# B&R Automation Studio project 8238 (part 17)

#### _GetRights.st - Ermittelt Lese- und Schreibrecht
```iecst
(********************************************************************
 * COPYRIGHT -- Herbert Kannegiesser GmbH
 ********************************************************************
 * Program: mnParam
 * File: _GetRights.st
 * Author: hunholz
 * Created: February 20, 2012
 ********************************************************************
 * Implementation of program mnParam
 ********************************************************************)

(* Ermittelt Lese- und Schreibrecht *)
FUNCTION_BLOCK _GetRights

	IF Enable THEN

		Status := ERR_OK;

		bWriteAccess := 0;
		bReadAccess := 0;

		IF lPtrLogicStruct = 0 THEN

			Status := MNPARAM_STAT_NULLPOINTER;
			RETURN;

		END_IF

		_DoLogStruc ACCESS lPtrLogicStruct;

		IF siWriteAccess >= 0 THEN

			bWriteAccess := SINT_TO_USINT(siWriteAccess);

		ELSE

			_wLogIdx := wReference;
			_xReady := FALSE;
			_bSearchIt := 0;

			REPEAT

				IF _wLogIdx <= wMaxIdxLogicStruct  AND _wLogIdx > 0 THEN

					IF _DoLogStruc.LogicalStruct[_wLogIdx].siWriteAccess >= 0 THEN

						// Gültiges Recht gefunden
						bWriteAccess := SINT_TO_USINT(_DoLogStruc.LogicalStruct[_wLogIdx].siWriteAccess);
						_xReady := TRUE;

					ELSE

						IF _DoLogStruc.LogicalStruct[_wLogIdx].iReferenz > 0 THEN

							_wLogIdx := INT_TO_UINT(_DoLogStruc.LogicalStruct[_wLogIdx].iReferenz);
							_bSearchIt := _bSearchIt + 1;

							// Wenn maximale Suchtiefe erreicht, dann abbrechen
							_xReady := _bSearchIt > 6;

						ELSE

							// Kein Recht definiert und Referenz verweist auf Container, abbrechen
							_xReady := TRUE;

						END_IF

					END_IF

				ELSE

					// Referenz ist ungültig, abbrechen
					_xReady := TRUE;

				END_IF

				UNTIL
					_xReady
			END_REPEAT

		END_IF

		IF siReadAccess >= 0 THEN

			bReadAccess := SINT_TO_USINT(siReadAccess);

		ELSE

			_wLogIdx := wReference;
			_xReady := FALSE;
			_bSearchIt := 0;

			REPEAT

				IF _wLogIdx <= wMaxIdxLogicStruct  AND _wLogIdx > 0 THEN

					IF _DoLogStruc.LogicalStruct[_wLogIdx].siVisibleAccess >= 0 THEN

						// Gültiges Recht gefunden
						bReadAccess := SINT_TO_USINT(_DoLogStruc.LogicalStruct[_wLogIdx].siVisibleAccess);
						_xReady := TRUE;

					ELSE

						IF _DoLogStruc.LogicalStruct[_wLogIdx].iReferenz > 0 THEN

							_wLogIdx := INT_TO_UINT(_DoLogStruc.LogicalStruct[_wLogIdx].iReferenz);
							_bSearchIt := _bSearchIt + 1;

							// Wenn maximale Suchtiefe erreicht, dann abbrechen
							_xReady := _bSearchIt > 6;

						ELSE

							// Kein Recht definiert und Referenz verweist auf Container, abbrechen
							_xReady := TRUE;

						END_IF

					END_IF

				ELSE

					// Referenz ist ungültig, abbrechen
					_xReady := TRUE;

				END_IF

				UNTIL
				_xReady
			END_REPEAT

		END_IF

	ELSE

		Status := ERR_FUB_ENABLE_FALSE;

	END_IF

END_FUNCTION_BLOCK
```

#### _BinSearchTxtLine.st - Finde Textzeile nach Function-ID und Nummer
```iecst
(********************************************************************
 * COPYRIGHT -- Herbert Kannegiesser GmbH
 ********************************************************************
 * Program: mnParam
 * File: _BinSearchTxtLine.st
 * Author: hunholz
 * Created: February 21, 2012
 ********************************************************************
 * Implementation of program mnParam
 ********************************************************************)

(* Finde Textzeile nach Function-ID und Nummer *)
FUNCTION _BinSearchTxtLine

	_BinSearchTxtLine := 65535;

	IF lPtrTxtLines = 0 OR wCntRows < 1 THEN
		// Null-Pointer oder leere Liste
		RETURN;
	END_IF

	// Access auf dynamische Struktur
	_pTextLines ACCESS lPtrTxtLines;

	_wMin := 0;
	_wMax := wCntRows-1;

	WHILE TRUE DO

		IF (_wMin <= _wMax) THEN

			// Suche nach korrektem IdxPar
			// Middle Index berechnen
			_wMid := (_wMin + _wMax) / 2;

			// Suche erfolgreich?
			IF _pTextLines[_wMid].wFunctionID = wFunctionID THEN

				IF _pTextLines[_wMid].wNumber = wNo THEN

					_BinSearchTxtLine := _wMid;

					EXIT;

				ELSIF wNo < _pTextLines[_wMid].wNumber THEN

					_wMax := _wMid - 1;

				ELSE

					_wMin := _wMid + 1;

				END_IF

			ELSIF wFunctionID < _pTextLines[_wMid].wFunctionID THEN

				_wMax := _wMid - 1;

			ELSE

				_wMin := _wMid + 1;

			END_IF

		ELSE
			// Fehler in der Binären-Suche
			// zB entsprechende Zeile konnte nicht gefunden werden
			EXIT;
		END_IF;

	END_WHILE;

END_FUNCTION
```

#### _BinSearchHlpTxtLine.st - Finde Hilfstextzeile nach Funktion-ID und Nummer
```iecst
(********************************************************************
 * COPYRIGHT -- Herbert Kannegiesser GmbH
 ********************************************************************
 * Program: mnParam
 * File: _BinSearchHlpTxtLine.st
 * Author: hunholz
 * Created: February 21, 2012
 ********************************************************************
 * Implementation of program mnParam
 ********************************************************************)

(* Finde Hilfstextzeile nach Funktion-ID und Nummer *)
FUNCTION _BinSearchHlpTxtLine

	_BinSearchHlpTxtLine := 65535;

	IF lPtrHlpTxtLines = 0 OR wCntRows < 1 THEN
		// Null-Pointer oder leere Liste
		RETURN;
	END_IF

	// Access auf dynamische Struktur
	_pHlpTextLines ACCESS lPtrHlpTxtLines;

	_wMin := 0;
	_wMax := wCntRows-1;

	WHILE TRUE DO

		IF (_wMin <= _wMax) THEN

			// Suche nach korrektem IdxPar
			// Middle Index berechnen
			_wMid := (_wMin + _wMax) / 2;

			// Suche erfolgreich?
			IF _pHlpTextLines[_wMid].wFunctionID = wFunctionID THEN

				IF _pHlpTextLines[_wMid].wNumber = wNo THEN

					_BinSearchHlpTxtLine := _wMid;

					EXIT;

				ELSIF wNo < _pHlpTextLines[_wMid].wNumber THEN

					_wMax := _wMid - 1;

				ELSE

					_wMin := _wMid + 1;

				END_IF

			ELSIF wFunctionID < _pHlpTextLines[_wMid].wFunctionID THEN

				_wMax := _wMid - 1;

			ELSE

				_wMin := _wMid + 1;

			END_IF

		ELSE
			// Fehler in der Binären-Suche
			// zB entsprechende Zeile konnte nicht gefunden werden
			EXIT;
		END_IF;

	END_WHILE;

END_FUNCTION
```

#### _LimParam.st - Parameter begrenzen
```iecst
(********************************************************************
 * COPYRIGHT -- Herbert Kannegiesser GmbH
 ********************************************************************
 * Program: mnParam
 * File: _LimParam.st
 * Author: hunholz
 * Created: June 12, 2012
 ********************************************************************
 * Implementation of program mnParam
 ********************************************************************)

(* Parameter begrenzen *)
FUNCTION_BLOCK _LimParam

	IF pParamNum = 0 OR pCsvNumRow = 0 THEN

		RETURN;

	END_IF

	_ParamNum ACCESS pParamNum;
	_CsvNumRow ACCESS pCsvNumRow;

	IF _CsvNumRow.bRowType = 10 THEN

		_CsvNumRow.diValue := LIMIT(_ParamNum.diMinValue, _CsvNumRow.diValue, _ParamNum.diMaxValue);

	ELSE

		_rValue ACCESS ADR(_CsvNumRow.diValue);
		_rMinValue ACCESS ADR(_ParamNum.diMinValue);
		_rMaxValue ACCESS ADR(_ParamNum.diMaxValue);

		_rValue := LIMIT(_rMinValue, _rValue, _rMaxValue);

	END_IF

END_FUNCTION_BLOCK
```

#### mnParam.fun
```iecst
(********************************************************************
 * COPYRIGHT -- Herbert Kannegiesser GmbH
 ********************************************************************
 * Program: mnParam
 * File: mnParam.fun
 * Author: hunholz
 * Created: February 16, 2012
 ********************************************************************
 * Functions and function blocks of program mnParam
 ********************************************************************)

FUNCTION_BLOCK _ExportContainer (*Schreibe Containerdaten in eine CSV-Datei*)
	VAR_INPUT
		Enable : BOOL;
		pIntern : UDINT;
	END_VAR
	VAR_OUTPUT
		Status : UINT;
		AdStatus : UINT;
		dtContainerWritten : DATE_AND_TIME;
	END_VAR
	VAR
		_Intern : REFERENCE TO PmIntern_typ;
		_ContainerExpState : enum_ContainerExportState := ces_AllocMemCSV;
		_xBusy : BOOL;
		_xReady : BOOL;
		_MemPartAlloc : AsMemPartAllocClear;
		_wIntStatus : UINT;
		_WriteBOM : mnParam_WriteBOM_Mem;
		_WriteComment : mnParam_WriteCSV254_Mem;
		_WriteNewLine : mnParam_WriteNewline_Mem;
		_WriteFileEnd : mnParam_WriteCSV255_Mem;
		_WriteVersion : mnParam_WriteCSV253_Mem;
		_WriteMachineNo : mnParam_WriteCSV252_Mem;
		_WriteTimeStamp : mnParam_WriteCSV251_Mem;
		_WriteNumPar : mnParam_WriteCSV10_Mem;
		_WriteRealPar : mnParam_WriteCSV11_Mem;
		_WriteString : mnParam_WriteCSV20_Mem;
		_DoContainer : REFERENCE TO mnParam_ContainerDyn_typ;
		_DoParamNum : REFERENCE TO mnParam_ParamNumDyn_typ;
		_DoParamString : REFERENCE TO mnParam_ParamStringDyn_typ;
		_DoNum : REFERENCE TO mnParam_CsvNumDyn_typ;
		_DoString : REFERENCE TO mnParam_CsvStringDyn_typ;
		_wOldIdx : UINT;
		_i : UINT;
		_deleteCSVFile : FileDelete;
		_createCSVFile : FileCreate;
		_openCSVFile : FileOpen;
		_writeCSVFile : FileWrite;
		_DTGetTime : DTGetTime;
		_xFault : BOOL;
		_closeCSVFile : FileClose;
		_wIntAdStatus : UINT;
		_MemPartFree : AsMemPartFree;
		_sPathAndFilename : STRING[63];
		_wIdxToc : UINT;
	END_VAR
END_FUNCTION_BLOCK

FUNCTION_BLOCK _ExportToc (*Inhaltsverzeichnis schreiben*)
	VAR_INPUT
		Enable : BOOL;
		pIntern : UDINT;
	END_VAR
	VAR_OUTPUT
		Status : UINT;
		AdStatus : UINT;
		dtTocWritten : DATE_AND_TIME;
	END_VAR
	VAR
		_Intern : REFERENCE TO PmIntern_typ;
		_xReady : BOOL;
		_xBusy : BOOL;
		_TocExpState : enum_TocExportState;
		_wIntStatus : UINT;
		_MemPartAlloc : AsMemPartAllocClear;
		_xFault : BOOL;
		_WriteToc : mnParam_WriteCSV80_Mem;
		_i : UINT;
		_WriteBOM : mnParam_WriteBOM_Mem;
		_WriteComment : mnParam_WriteCSV254_Mem;
		_WriteNewLine : mnParam_WriteNewline_Mem;
		_WriteVersion : mnParam_WriteCSV253_Mem;
		_WriteMachineNo : mnParam_WriteCSV252_Mem;
		_WriteTimeStamp : mnParam_WriteCSV251_Mem;
		_DTGetTime : DTGetTime;
		_HeaderTimeRow : mnParam_HeaderTimeRow_typ;
		_sPathAndFilename : STRING[63];
		_deleteCSVFile : FileDelete;
		_WriteFileEnd : mnParam_WriteCSV255_Mem;
		_createCSVFile : FileCreate;
		_wIntAdStatus : UINT;
		_openCSVFile : FileOpen;
		_writeCSVFile : FileWrite;
		_closeCSVFile : FileClose;
		_MemPartFree : AsMemPartFree;
	END_VAR
END_FUNCTION_BLOCK

FUNCTION_BLOCK _DefActContainer (*Fülle ActContainer*)
	VAR_INPUT
		Enable : BOOL;
		bContainerIdx : USINT;
		wInstanceIdx : UINT;
		pIntern : UDINT;
	END_VAR
	VAR_OUTPUT
		Status : UINT;
	END_VAR
	VAR
		_Intern : REFERENCE TO PmIntern_typ;
		_DoContainer : REFERENCE TO mnParam_ContainerDyn_typ;
		_lPVadress : UDINT;
		_lPVlen : UDINT;
		_wDimension : UINT;
		_sIndex : STRING[5];
	END_VAR
END_FUNCTION_BLOCK

FUNCTION_BLOCK _GetRights (*Ermittelt Lese- und Schreibrecht*)
	VAR_INPUT
		Enable : BOOL;
		siWriteAccess : SINT;
		siReadAccess : SINT;
		wReference : UINT;
		lPtrLogicStruct : UDINT;
		wMaxIdxLogicStruct : UINT;
	END_VAR
	VAR_OUTPUT
		bWriteAccess : USINT;
		bReadAccess : USINT;
		Status : UINT;
	END_VAR
	VAR
		_DoLogStruc : REFERENCE TO mnParam_LogicalStructDyn_typ;
		_wLogIdx : UINT;
		_xReady : BOOL;
		_bSearchIt : USINT;
	END_VAR
END_FUNCTION_BLOCK

FUNCTION _BinSearchTxtLine : UINT (*Finde Textzeile nach Function-ID und Nummer*)
	VAR_INPUT
		wFunctionID : UINT;
		wNo : UINT;
		lPtrTxtLines : UDINT;
		wCntRows : UINT;
	END_VAR
	VAR
		_pTextLines : REFERENCE TO ARRAY[0..65534] OF mnTxt_TxtLine_Typ;
		_wMin : UINT;
		_wMax : UINT;
		_wMid : UINT;
	END_VAR
END_FUNCTION

FUNCTION _BinSearchHlpTxtLine : UINT (*Finde Hilfstextzeile nach Funktion-ID und Nummer*)
	VAR_INPUT
		wFunctionID : UINT;
		wNo : UINT;
		lPtrHlpTxtLines : UDINT;
		wCntRows : UINT;
	END_VAR
	VAR
		_pHlpTextLines : REFERENCE TO ARRAY[0..65534] OF mnTxt_HelpTxtLine_Typ;
		_wMin : UINT;
		_wMax : UINT;
		_wMid : UINT;
	END_VAR
END_FUNCTION

FUNCTION_BLOCK _LimParam (*Parameter begrenzen*)
	VAR_INPUT
		pCsvNumRow : UDINT;
		pParamNum : UDINT;
	END_VAR
	VAR
		_ParamNum : REFERENCE TO mnParam_ParamNumRow_typ;
		_CsvNumRow : REFERENCE TO mnParam_CsvNumRow_typ;
		_rValue : REFERENCE TO REAL;
		_rMinValue : REFERENCE TO REAL;
		_rMaxValue : REFERENCE TO REAL;
	END_VAR
END_FUNCTION_BLOCK
```

#### _actInterfacePC.st
```iecst
(********************************************************************
 * COPYRIGHT -- Herbert Kannegiesser GmbH
 ********************************************************************
 * Program: mnParam
 * File: _actInterfacePC.st
 * Author: hunholz
 * Created: March 28, 2012
 ********************************************************************
 * Implementation of program mnParam
 ********************************************************************)

(* Kommando-Interface zum PC über mnParamCmd *)
ACTION _actInterfacePC:

	CASE _PmIntern.enCycMainState OF

		cs_MainIdle:

			//************************************************
			// Kein PC-Befehl aktiv. Warte auf Befehl
			//************************************************

			CASE mnParamCmd.Request.Command.wCommand OF

				MNPARAM_CMD_NOCOMMAND:

					mnParamCmd.Response.wCmdStatus := MNPARAM_STAT_NOCOMMAND;

				MNPARAM_CMD_IMPORT:

					IF _xAllowCommands THEN

						_xAllowCommands := FALSE;

						// Warten bis Import abgeschlossen
						_PmIntern.enCycMainState := cs_MainImport;

						// Wir MNPARAM_IMPORT_RESTORE als Attribut mitgegeben, werden vor dem Import
						// alle Variablen auf Default gesetzt.
						_wImpSource := UDINT_TO_UINT(mnParamCmd.Request.Command.lData0);
						_xImpSetDefault := mnParamCmd.Request.Command.lData1 = MNPARAM_IMPORT_RESTORE;

						mnParamCmd.Response.wCmdStatus := KG_STAT_BUSY;

						_LogEntryIn.wErrorNo := _MNPARAM_LOG_STARTIMPORT;
						_LogEntryIn.lAttr1 := mnParamCmd.Request.Command.lData0;
						_LogEntryIn.lAttr2 := mnParamCmd.Request.Command.lData1;
						_InsertRB(wPtrStart := _wPtrRBstart, wPtrRead := _wPtrRBread, wPtrWrite := _wPtrRBwrite);

						// Starte Import
						_PmIntern.enCycImpState := cs_ImpStart;

					ELSE

						// Kommando ablehnen
						mnParamCmd.Response.wCmdStatus := KG_CMDSTAT_NOTREADY;
						_PmIntern.enCycMainState := cs_MainWaitCmdZero;

					END_IF

				MNPARAM_CMD_DELETE:

					IF _xAllowCommands THEN

						_xAllowCommands := FALSE;

						// Warten bis Delete abgeschlossen
						_PmIntern.enCycMainState := cs_MainDelete;

						// Parameter übernehmen
						_wDelCont := UDINT_TO_UINT(mnParamCmd.Request.Command.lData0);
						_wDelInst := UDINT_TO_UINT(mnParamCmd.Request.Command.lData1);

						mnParamCmd.Response.wCmdStatus := KG_STAT_BUSY;

						_LogEntryIn.wErrorNo := _MNPARAM_LOG_STARTDELETE;
						_LogEntryIn.lAttr1 := mnParamCmd.Request.Command.lData0;
						_LogEntryIn.lAttr2 := mnParamCmd.Request.Command.lData1;
						_InsertRB(wPtrStart := _wPtrRBstart, wPtrRead := _wPtrRBread, wPtrWrite := _wPtrRBwrite);

						// Starte Delete
						_PmIntern.enCycDelState := cs_DelStart;

					ELSE

						// Kommando ablehnen
						mnParamCmd.Response.wCmdStatus := KG_CMDSTAT_NOTREADY;
						_PmIntern.enCycMainState := cs_MainWaitCmdZero;

					END_IF

				ELSE
					// ungültiges Kommando
					mnParamCmd.Response.wCmdStatus := KG_CMDSTAT_NOTVALID;
					_PmIntern.enCycMainState := cs_MainWaitCmdZero;

			END_CASE

		cs_MainImport:

			mnParamCmd.Response.wCmdStatus := KG_STAT_BUSY;

			// Warten bis Import fertig ist
			IF _PmIntern.enCycImpState = cs_ImpRdySuccess THEN

				// ERFOLG

				// Import Statemachine zurücksetzen
				_PmIntern.enCycImpState := cs_ImpIdle;

				// Rückmeldung OK
				mnParamCmd.Response.wCmdStatus := MNPARAM_CMD_IMPORT;

				_LogEntryIn.wErrorNo := _MNPARAM_LOG_ENDIMPORT_SUCC;
				_InsertRB(wPtrStart := _wPtrRBstart, wPtrRead := _wPtrRBread, wPtrWrite := _wPtrRBwrite);

				_actFillNamelist;

				_PmIntern.enCycMainState := cs_MainWaitCmdZero;

			ELSIF _PmIntern.enCycImpState = cs_ImpRdyFault THEN

				// FEHLER

				// Import Statemachine zurücksetzen
				_PmIntern.enCycImpState := cs_ImpIdle;

				// Fehlercode für Rückmeldung übernehmen
				mnParamCmd.Response.wCmdStatus := MAX(59999,DINT_TO_UINT(_PmIntern.Status.diMsgAttr1));

				_LogEntryIn.wErrorNo := _MNPARAM_LOG_ENDIMPORT_FAILED;
				_LogEntryIn.lAttr1 := mnParamCmd.Response.wCmdStatus;
				_InsertRB(wPtrStart := _wPtrRBstart, wPtrRead := _wPtrRBread, wPtrWrite := _wPtrRBwrite);

				// Warnung ausgeben
				_PmIntern.enCycMainState := cs_MainWarning;

			END_IF

		cs_MainDelete:

			mnParamCmd.Response.wCmdStatus := KG_STAT_BUSY;

			// Warten bis Delete fertig ist
			IF _PmIntern.enCycDelState = cs_DelRdySuccess THEN

				// ERFOLG

				// Delete Statemachine zurücksetzen
				_PmIntern.enCycDelState := cs_DelIdle;

				// Rückmeldung OK
				mnParamCmd.Response.wCmdStatus := MNPARAM_CMD_DELETE;

				_LogEntryIn.wErrorNo := _MNPARAM_LOG_ENDDELETE_SUCC;
				_InsertRB(wPtrStart := _wPtrRBstart, wPtrRead := _wPtrRBread, wPtrWrite := _wPtrRBwrite);

				IF _wDelCont = MNPARAM_IDX_PROGCONTAINER THEN

					_actFillNamelist;

				END_IF

				_PmIntern.enCycMainState := cs_MainWaitCmdZero;

			ELSIF _PmIntern.enCycDelState = cs_DelRdyFault THEN

				// FEHLER

				// Delete Statemachine zurücksetzen
				_PmIntern.enCycDelState := cs_DelIdle;

				// Fehlercode als Rückmeldung
				mnParamCmd.Response.wCmdStatus := MAX(59999,DINT_TO_UINT(_PmIntern.Status.diMsgAttr1));

				_LogEntryIn.wErrorNo := _MNPARAM_LOG_ENDDELETE_FAILED;
				_LogEntryIn.lAttr1 := mnParamCmd.Response.wCmdStatus;
				_InsertRB(wPtrStart := _wPtrRBstart, wPtrRead := _wPtrRBread, wPtrWrite := _wPtrRBwrite);

				// Warnung ausgeben
				_PmIntern.enCycMainState := cs_MainWarning;

			END_IF

		cs_MainWarning:

			//*****************
			// Warnung ausgeben
			//*****************

			mnParamCmd.Response.wCmdStatus := MAX(59999,DINT_TO_UINT(_PmIntern.Status.diMsgAttr1));

			IF TONwarn.Q THEN

				// Warnungszeit ist abgelaufen

				// Warnung zurücksetzen
				brsmemset(ADR(_PmIntern.Status), 0, SIZEOF(_PmIntern.Status));
				_PmIntern.Status.wFunction_ID := MNPARAM_FUNCTIONID;

				// Auf Rücksetzen des Kommandos warten
				_PmIntern.enCycMainState := cs_MainWaitCmdZero;

			END_IF

		cs_MainWaitCmdZero:

			//**********************************************
			// Warten, dass das Kommando zurückgenommen wird
			//**********************************************

			IF mnParamCmd.Request.Command.wCommand = MNPARAM_CMD_NOCOMMAND THEN

				mnParamCmd.Response.wCmdStatus := MNPARAM_STAT_NOCOMMAND;
				_PmIntern.enCycMainState := cs_MainIdle;

			END_IF

	END_CASE

	// Warnung soll für 10 Sekunden anstehen
	TONwarn(IN := _PmIntern.enCycMainState = cs_MainWarning, PT := T#10s);

END_ACTION
```

#### _actInterfaceApplication.st
```iecst
(********************************************************************
 * COPYRIGHT -- Herbert Kannegiesser GmbH
 ********************************************************************
 * Program: mnParam
 * File: _actInterfaceApplication.st
 * Author: hunholz
 * Created: March 28, 2012
 ********************************************************************
 * Implementation of program mnParam
 ********************************************************************)

(* Kommando-Interface zur Applikation über IFmnParam *)
ACTION _actInterfaceApplication:

	CASE _PmIntern.enCycIfState OF

		cs_IfIdle:

			//*************************************************
			// Kein Applikations-Befehl aktiv. Warte auf Befehl
			//*************************************************

			CASE IFmnParam.In.Edit.wCommand OF

				MNPARAM_CMD_NOCOMMAND:

					IFmnParam.Out.Edit.wStatus := MNPARAM_STAT_NOCOMMAND;

				MNPARAM_CMD_FILLEDITOR:

					IF _xAllowCommands THEN

						_xAllowCommands := FALSE;

						// Warten bis das Füllen des Editors abgeschlossen ist.
						_PmIntern.enCycIfState := cs_IfFillEditor;

						IFmnParam.Out.Edit.wStatus := KG_CMDSTAT_BUSY;

						// Füllen des Editors starten
						_PmIntern.enCycFillEditor := cs_feStart;

					ELSE

						// Kommando ablehnen
						IFmnParam.Out.Edit.wStatus := KG_CMDSTAT_NOTREADY;
						// Kommando muss zurückgenommen werden
						_PmIntern.enCycIfState := cs_IfReady;

					END_IF

				MNPARAM_CMD_SAVEEDITOR:

					IF _xAllowCommands THEN

						_xAllowCommands := FALSE;

						// Warten bis das Sichern des Editors abgeschlossen ist
						_PmIntern.enCycIfState := cs_IfSaveEditor;

						IFmnParam.Out.Edit.wStatus := KG_CMDSTAT_BUSY;

						_LogEntryIn.wErrorNo := _MNPARAM_LOG_STARTSAVE;
						_InsertRB(wPtrStart := _wPtrRBstart, wPtrRead := _wPtrRBread, wPtrWrite := _wPtrRBwrite);

						// Sichern starten
						_PmIntern.enCycSaveEditor := cs_seStart;

					ELSE

						// Kommando ablehnen
						IFmnParam.Out.Edit.wStatus := KG_CMDSTAT_NOTREADY;
						// Kommando muss zurückgenommen werden
						_PmIntern.enCycIfState := cs_IfReady;

					END_IF

				MNPARAM_CMD_CREATE_INDCONT:

					IF _xAllowCommands THEN

						_xAllowCommands := FALSE;

						// Parameter übernehmen
						_wCreateCont := IFmnParam.In.Edit.bContainer;

						IF IFmnParam.In.Edit.diContainerInstance < 0 THEN

							IF _wCreateCont <= MNPARAM_MAXIDX_CONTAINER THEN

								IF _pDoContainer.Container[_wCreateCont].bDirectParam = 0 THEN

									FOR _inst := 0 TO _pDoContainer.Container[_wCreateCont].wDimension - 1 DO

										IF NOT(_PmIntern.TOC.TocEntry[_PmIntern.TOC.wStartIdx[_wCreateCont] + _inst].xExist) THEN
											EXIT;
										END_IF

									END_FOR

									IF _inst < _pDoContainer.Container[_wCreateCont].wDimension THEN

										_wCreateInst := _pDoContainer.Container[_wCreateCont].wMinBound + _inst;

										// Warten bis das Anlegen einer Instanz abgeschlossen ist
										_PmIntern.enCycIfState := cs_IfCreateIndCont;

										IFmnParam.Out.Edit.wStatus := KG_CMDSTAT_BUSY;

										_LogEntryIn.wErrorNo := _MNPARAM_LOG_STARTCREATE;
										_LogEntryIn.lAttr1 := _wCreateCont;
										_LogEntryIn.lAttr2 := _wCreateInst;
										_InsertRB(wPtrStart := _wPtrRBstart, wPtrRead := _wPtrRBread, wPtrWrite := _wPtrRBwrite);

										// Instanz anlegen
										_PmIntern.enCycCreate := cs_CrtStart;

									ELSE

										// Warten bis das Anlegen einer Instanz abgeschlossen ist
										_PmIntern.enCycIfState := cs_IfReady;
										IFmnParam.Out.Edit.wStatus := MNPARAM_STAT_NO_FREE_CONTINST;

									END_IF

								ELSE

									// Warten bis das Anlegen einer Instanz abgeschlossen ist
									_PmIntern.enCycIfState := cs_IfReady;
									IFmnParam.Out.Edit.wStatus := MNPARAM_STAT_CONTAINER_NOT_VALID;

								END_IF

							ELSE

								// Warten bis das Anlegen einer Instanz abgeschlossen ist
								_PmIntern.enCycIfState := cs_IfReady;
								IFmnParam.Out.Edit.wStatus := MNPARAM_STAT_CONTAINER_NOT_VALID;

							END_IF

						ELSE

							_wCreateInst := DINT_TO_UINT(IFmnParam.In.Edit.diContainerInstance);

							// Warten bis das Anlegen einer Instanz abgeschlossen ist
							_PmIntern.enCycIfState := cs_IfCreateIndCont;

							IFmnParam.Out.Edit.wStatus := KG_CMDSTAT_BUSY;

							_LogEntryIn.wErrorNo := _MNPARAM_LOG_STARTCREATE;
							_LogEntryIn.lAttr1 := _wCreateCont;
							_LogEntryIn.lAttr2 := _wCreateInst;
							_InsertRB(wPtrStart := _wPtrRBstart, wPtrRead := _wPtrRBread, wPtrWrite := _wPtrRBwrite);

							// Instanz anlegen
							_PmIntern.enCycCreate := cs_CrtStart;

						END_IF

					ELSE

						// Kommando ablehnen
						IFmnParam.Out.Edit.wStatus := KG_CMDSTAT_NOTREADY;
						// Kommando muss zurückgenommen werden
						_PmIntern.enCycIfState := cs_IfReady;

					END_IF

				MNPARAM_CMD_DELETE_INDCONT:

					IF _xAllowCommands THEN

						_xAllowCommands := FALSE;

						// Warten bis das Löschen der Instanz abgeschlossen ist
						_PmIntern.enCycIfState := cs_IfDeleteIndCont;

						IFmnParam.Out.Edit.wStatus := KG_CMDSTAT_BUSY;

						// Parameter übernehmen
						_wDelCont := IFmnParam.In.Edit.bContainer;
						_wDelInst := DINT_TO_UINT(IFmnParam.In.Edit.diContainerInstance);

						_LogEntryIn.wErrorNo := _MNPARAM_LOG_STARTDELETE;
						_LogEntryIn.lAttr1 := _wDelCont;
						_LogEntryIn.lAttr2 := _wDelInst;
						_InsertRB(wPtrStart := _wPtrRBstart, wPtrRead := _wPtrRBread, wPtrWrite := _wPtrRBwrite);

						// Löschen starten
						_PmIntern.enCycDelState := cs_DelStart;

					ELSE

						// Kommando ablehnen
						IFmnParam.Out.Edit.wStatus := KG_CMDSTAT_NOTREADY;
						// Kommando muss zurückgenommen werden
						_PmIntern.enCycIfState := cs_IfReady;

					END_IF

				MNPARAM_CMD_COPY_INDCONT:

					IF _xAllowCommands THEN

						_xAllowCommands := FALSE;

						// Parameter übernehmen
						_wCopyCont := IFmnParam.In.Edit.bContainer;
						_wCopyInstFrom := IFmnParam.In.Edit.wContainerInstanceFrom;

						IF IFmnParam.In.Edit.diContainerInstance < 0 THEN

							IF _wCopyCont <= MNPARAM_MAXIDX_CONTAINER THEN

								IF _pDoContainer.Container[_wCopyCont].bDirectParam = 0 THEN

									FOR _inst := 0 TO _pDoContainer.Container[_wCopyCont].wDimension - 1 DO

										IF NOT(_PmIntern.TOC.TocEntry[_PmIntern.TOC.wStartIdx[_wCopyCont] + _inst].xExist) THEN
											EXIT;
										END_IF

									END_FOR

									IF _inst < _pDoContainer.Container[_wCopyCont].wDimension THEN

										_wCopyInst := _pDoContainer.Container[_wCopyCont].wMinBound + _inst;

										// Warten bis das Kopieren einer Instanz abgeschlossen ist
										_PmIntern.enCycIfState := cs_IfCopyIndCont;

										IFmnParam.Out.Edit.wStatus := KG_CMDSTAT_BUSY;

										_LogEntryIn.wErrorNo := _MNPARAM_LOG_STARTCOPY;
										_LogEntryIn.lAttr1 := _wCreateCont;
										_LogEntryIn.lAttr2 := _wCreateInst;
										_InsertRB(wPtrStart := _wPtrRBstart, wPtrRead := _wPtrRBread, wPtrWrite := _wPtrRBwrite);

										// Instanz anlegen
										_PmIntern.enCycCopy := cs_CpyStart;

									ELSE

										// Warten bis das Anlegen einer Instanz abgeschlossen ist
										_PmIntern.enCycIfState := cs_IfReady;
										IFmnParam.Out.Edit.wStatus := MNPARAM_STAT_NO_FREE_CONTINST;

									END_IF

								ELSE

									// Warten bis das Anlegen einer Instanz abgeschlossen ist
									_PmIntern.enCycIfState := cs_IfReady;
									IFmnParam.Out.Edit.wStatus := MNPARAM_STAT_CONTAINER_NOT_VALID;

								END_IF

							ELSE

								// Warten bis das Anlegen einer Instanz abgeschlossen ist
								_PmIntern.enCycIfState := cs_IfReady;
								IFmnParam.Out.Edit.wStatus := MNPARAM_STAT_CONTAINER_NOT_VALID;

							END_IF

						ELSE

							_wCopyInst := DINT_TO_UINT(IFmnParam.In.Edit.diContainerInstance);

							// Warten bis das Kopieren einer Instanz abgeschlossen ist
							_PmIntern.enCycIfState := cs_IfCopyIndCont;

							IFmnParam.Out.Edit.wStatus := KG_CMDSTAT_BUSY;

							_LogEntryIn.wErrorNo := _MNPARAM_LOG_STARTCOPY;
							_LogEntryIn.lAttr1 := _wCreateCont;
							_LogEntryIn.lAttr2 := _wCreateInst;
							_InsertRB(wPtrStart := _wPtrRBstart, wPtrRead := _wPtrRBread, wPtrWrite := _wPtrRBwrite);

							// Instanz anlegen
							_PmIntern.enCycCopy := cs_CpyStart;

						END_IF

					ELSE

						// Kommando ablehnen
						IFmnParam.Out.Edit.wStatus := KG_CMDSTAT_NOTREADY;
						// Kommando muss zurückgenommen werden
						_PmIntern.enCycIfState := cs_IfReady;

					END_IF

				MNPARAM_CMD_BACKUP:

					IF _xAllowCommands THEN

						_xAllowCommands := FALSE;

						// USB-Flashdisk muss gesteckt sein
						IF IFmnSystem.Out.xUSBStickReady THEN

							// Warten bis Backup beendet ist
							_PmIntern.enCycIfState := cs_IfBackup;

							IFmnParam.Out.Edit.wStatus := KG_CMDSTAT_BUSY;

							_LogEntryIn.wErrorNo := _MNPARAM_LOG_STARTBACKUP;
							_LogEntryIn.lAttr1 := 0;
							_LogEntryIn.lAttr2 := 0;
							_InsertRB(wPtrStart := _wPtrRBstart, wPtrRead := _wPtrRBread, wPtrWrite := _wPtrRBwrite);

							// Devicenamen der USB-Flashdisk übernehmen
							_sUSBInterface := IFmnSystem.Out.sInterfaceUSB;

							// Backup starten
							_PmIntern.enCycBackup := cs_BacUSBlinkDevice;

						ELSE

							// Es ist keine USB-Flashdisk gesteckt
							IFmnParam.Out.Edit.wStatus := MNPARAM_STAT_NOUSBSTICK;
							// Kommando muss zurückgenommen werden
							_PmIntern.enCycIfState := cs_IfReady;

						END_IF

					ELSE

						// Kommando ablehnen
						IFmnParam.Out.Edit.wStatus := KG_CMDSTAT_NOTREADY;
						// Kommando muss zurückgenommen werden
						_PmIntern.enCycIfState := cs_IfReady;

					END_IF

				MNPARAM_CMD_RESTORE:

					IF _xAllowCommands THEN

						_xAllowCommands := FALSE;

						// USB-Flashdisk muss gesteckt sein
						IF IFmnSystem.Out.xUSBStickReady THEN

							// Warten bis Restore abgeschlossen ist
							_PmIntern.enCycIfState := cs_IfRestore;

							IFmnParam.Out.Edit.wStatus := KG_CMDSTAT_BUSY;

							// Devicenamen der USB-Flashdisk übernehmen
							_sUSBInterface := IFmnSystem.Out.sInterfaceUSB;

							_LogEntryIn.wErrorNo := _MNPARAM_LOG_STARTRESTORE;
							_LogEntryIn.lAttr1 := 0;
							_LogEntryIn.lAttr2 := 0;
							_InsertRB(wPtrStart := _wPtrRBstart, wPtrRead := _wPtrRBread, wPtrWrite := _wPtrRBwrite);

							// Restore starten
							_PmIntern.enCycImpState := cs_ImpUSBLinkDevice;

						ELSE

							// Es ist keine USB-Flashdisk gesteckt
							IFmnParam.Out.Edit.wStatus := MNPARAM_STAT_NOUSBSTICK;
							// Kommando muss zurückgenommen werden
							_PmIntern.enCycIfState := cs_IfReady;

						END_IF

					ELSE

						// Kommando ablehnen
						IFmnParam.Out.Edit.wStatus := KG_CMDSTAT_NOTREADY;
						// Kommando muss zurückgenommen werden
						_PmIntern.enCycIfState := cs_IfReady;

					END_IF

				MNPARAM_CMD_FILLNAMELIST:

					IF _xAllowCommands THEN

						_xAllowCommands := FALSE;

						IFmnParam.Out.Edit.wIdxContainerNamelist := IFmnParam.In.Edit.wSelIdxContainerNamelist;
						IFmnParam.Out.Edit.wParIdxNamelist := IFmnParam.In.Edit.wSelParIdxNamelist;

						_actFillNamelist;

						IFmnParam.Out.Edit.wStatus := KG_STAT_BUSY;

						_PmIntern.enCycIfState := cs_IfFillNameList;

					END_IF

				ELSE

					// Kommando ungültig
					IFmnParam.Out.Edit.wStatus := KG_CMDSTAT_NOTVALID;
					// Kommando muss zurückgenommen werden
					_PmIntern.enCycIfState := cs_IfReady;

			END_CASE

		cs_IfFillNameList:

			IF IFsvCPCache.In.wCmd = KG_CMD_NOCOMMAND AND IFsvCPCache.Out.wCmdResponse = KG_CMD_NOCOMMAND THEN

				IFsvCPCache.In.wSetOffset := 0;
				IFsvCPCache.In.wCmd := SVCPCACHE_CMD_SETOFFSET;

			END_IF

			IF IFsvCPCache.In.wCmd = SVCPCACHE_CMD_SETOFFSET AND IFsvCPCache.Out.wCmdResponse = SVCPCACHE_CMD_SETOFFSET THEN

				IFsvCPCache.In.wCmd := KG_CMD_NOCOMMAND;

				IFmnParam.Out.Edit.wStatus := MNPARAM_STAT_FILLNAMELIST_OK;
				_PmIntern.enCycIfState := cs_IfReady;

			END_IF

		cs_IfFillEditor:

			// Warten bis Füllen des Editor fertig ist
			IF _PmIntern.enCycFillEditor = cs_feRdySuccess THEN

				// ERFOLG

				// Rückmeldung
				IFmnParam.Out.Edit.wStatus := MNPARAM_STAT_FILLEDITOR_OK;

				// Statemachine Editor Füllen zurücksetzen
				_PmIntern.enCycFillEditor := cs_feIdle;
				// Kommando muss zurückgenommen werden
				_PmIntern.enCycIfState := cs_IfReady;

			ELSIF _PmIntern.enCycFillEditor = cs_feRdyFault THEN

				// FEHLER

				// Status zurückliefern
				IFmnParam.Out.Edit.wStatus := DINT_TO_UINT(_PmIntern.Status.diMsgAttr1);

				// Statemachine Editor Füllen zurücksetzen
				_PmIntern.enCycFillEditor := cs_feIdle;
				// Kommando muss zurückgenommen werden
				_PmIntern.enCycIfState := cs_IfReady;

			END_IF

		cs_IfSaveEditor:

			// Warten bis Editor gesichert wurde
			IF _PmIntern.enCycSaveEditor = cs_seRdySuccess THEN

				// ERFOLG

				// Rückmeldung
				IFmnParam.Out.Edit.wStatus := MNPARAM_STAT_SAVEEDITOR_OK;

				// Statemchine Editor sichern zurücksetzen
				_PmIntern.enCycSaveEditor := cs_seIdle;
				// Kommando muss zurückgenommen werden
				_PmIntern.enCycIfState := cs_IfReady;

				_LogEntryIn.wErrorNo := _MNPARAM_LOG_ENDSAVE_SUCC;
				_InsertRB(wPtrStart := _wPtrRBstart, wPtrRead := _wPtrRBread, wPtrWrite := _wPtrRBwrite);

			ELSIF _PmIntern.enCycSaveEditor = cs_seRdyFault THEN

				// FEHLER

				// Status zurückmelden
				IFmnParam.Out.Edit.wStatus := DINT_TO_UINT(_PmIntern.Status.diMsgAttr1);

				// Statemchine Editor sichern zurücksetzen
				_PmIntern.enCycSaveEditor := cs_seIdle;
				// Kommando muss zurückgenommen werden
				_PmIntern.enCycIfState := cs_IfReady;

				_LogEntryIn.wErrorNo := _MNPARAM_LOG_ENDSAVE_FAILED;
				_LogEntryIn.lAttr1 := IFmnParam.Out.Edit.wStatus;
				_InsertRB(wPtrStart := _wPtrRBstart, wPtrRead := _wPtrRBread, wPtrWrite := _wPtrRBwrite);

			END_IF

		cs_IfCreateIndCont:

			// Warten bis Instanz angelegt wurde
			IF _PmIntern.enCycCreate = cs_CrtRdySuccess THEN

				// ERFOLG

				// Rückmeldung
				IFmnParam.Out.Edit.wStatus := MNPARAM_STAT_CREATE_INDCONT_OK;

				// Statemachine Instanz anlegen zurücksetzen
				_PmIntern.enCycCreate := cs_CrtIdle;
				// Kommando muss zurückgenommen werden
				_PmIntern.enCycIfState := cs_IfReady;

				_LogEntryIn.wErrorNo := _MNPARAM_LOG_ENDCREATE_SUCC;
				_InsertRB(wPtrStart := _wPtrRBstart, wPtrRead := _wPtrRBread, wPtrWrite := _wPtrRBwrite);

				IF _wCreateCont = MNPARAM_IDX_PROGCONTAINER THEN

					_actFillNamelist;

				END_IF

			ELSIF _PmIntern.enCycCreate = cs_CrtRdyFault THEN

				// FEHLER

				// Status zurückmelden
				IFmnParam.Out.Edit.wStatus := DINT_TO_UINT(_PmIntern.Status.diMsgAttr1);

				// Statemachine Instanz anlegen zurücksetzen
				_PmIntern.enCycCreate := cs_CrtIdle;
				// Kommando muss zurückgenommen werden
				_PmIntern.enCycIfState := cs_IfReady;

				_LogEntryIn.wErrorNo := _MNPARAM_LOG_ENDCREATE_FAILED;
				_LogEntryIn.lAttr1 := IFmnParam.Out.Edit.wStatus;
				_InsertRB(wPtrStart := _wPtrRBstart, wPtrRead := _wPtrRBread, wPtrWrite := _wPtrRBwrite);

			END_IF

		cs_IfDeleteIndCont:

			// Warten bis Instanz löschen fertig ist
			IF _PmIntern.enCycDelState = cs_DelRdySuccess THEN

				// ERFOLG

				// Rückmeldung
				IFmnParam.Out.Edit.wStatus := MNPARAM_STAT_DELETE_INDCONT_OK;

				// Statemachin Delete zurücksetzen
				_PmIntern.enCycDelState := cs_DelIdle;
				// Kommando muss zurückgenommen werden
				_PmIntern.enCycIfState := cs_IfReady;

				_LogEntryIn.wErrorNo := _MNPARAM_LOG_ENDDELETE_SUCC;
				_InsertRB(wPtrStart := _wPtrRBstart, wPtrRead := _wPtrRBread, wPtrWrite := _wPtrRBwrite);

				IF _wDelCont = MNPARAM_IDX_PROGCONTAINER THEN

					_actFillNamelist;

				END_IF

			ELSIF _PmIntern.enCycDelState = cs_DelRdyFault THEN

				// FEHLER

				// Status zurückmelden
				IFmnParam.Out.Edit.wStatus := MAX(59999,DINT_TO_UINT(_PmIntern.Status.diMsgAttr1));

				// Statemachin Delete zurücksetzen
				_PmIntern.enCycDelState := cs_DelIdle;
				// Kommando muss zurückgenommen werden
				_PmIntern.enCycIfState := cs_IfReady;

				_LogEntryIn.wErrorNo := _MNPARAM_LOG_ENDDELETE_FAILED;
				_LogEntryIn.lAttr1 := IFmnParam.Out.Edit.wStatus;
				_InsertRB(wPtrStart := _wPtrRBstart, wPtrRead := _wPtrRBread, wPtrWrite := _wPtrRBwrite);

			END_IF

		cs_IfCopyIndCont:

			// Warten bis Instanz kopiert wurde
			IF _PmIntern.enCycCopy = cs_CpyRdySuccess THEN

				// ERFOLG

				// Status zurückmelden
				IFmnParam.Out.Edit.wStatus := MNPARAM_STAT_COPY_INDCONT_OK;

				// Statemachine Kopieren zurücksetzen
				_PmIntern.enCycCopy := cs_CpyIdle;
				// Kommando muss zurückgenommen werden
				_PmIntern.enCycIfState := cs_IfReady;

				_LogEntryIn.wErrorNo := _MNPARAM_LOG_ENDCOPY_SUCC;
				_InsertRB(wPtrStart := _wPtrRBstart, wPtrRead := _wPtrRBread, wPtrWrite := _wPtrRBwrite);

				IF _wCopyCont = MNPARAM_IDX_PROGCONTAINER THEN

					_actFillNamelist;

				END_IF

			ELSIF _PmIntern.enCycCopy = cs_CpyRdyFault THEN

				// FEHLER

				// Status zurückmelden
				IFmnParam.Out.Edit.wStatus := DINT_TO_UINT(_PmIntern.Status.diMsgAttr1);

				// Statemachine Kopieren zurücksetzen
				_PmIntern.enCycCopy := cs_CpyIdle;
				// Kommando muss zurückgenommen werden
				_PmIntern.enCycIfState := cs_IfReady;

				_LogEntryIn.wErrorNo := _MNPARAM_LOG_ENDCOPY_FAILED;
				_LogEntryIn.lAttr1 := IFmnParam.Out.Edit.wStatus;
				_InsertRB(wPtrStart := _wPtrRBstart, wPtrRead := _wPtrRBread, wPtrWrite := _wPtrRBwrite);

			END_IF

		cs_IfBackup:

			// Warten bis Backup fertig ist
			IF _PmIntern.enCycBackup = cs_BacRdySuccess THEN

				// ERFOLG

				// Rückmeldung
				IFmnParam.Out.Edit.wStatus := MNPARAM_STAT_BACKUP_OK;

				// Statemachine Backup zurücksetzen
				_PmIntern.enCycBackup := cs_BacIdle;
				// Kommando muss zurückgenommen werden
				_PmIntern.enCycIfState := cs_IfReady;

				_LogEntryIn.wErrorNo := _MNPARAM_LOG_ENDBACKUP_SUCC;
				_InsertRB(wPtrStart := _wPtrRBstart, wPtrRead := _wPtrRBread, wPtrWrite := _wPtrRBwrite);

			ELSIF _PmIntern.enCycBackup = cs_BacRdyFault THEN

				// FEHLER

				// Status zurückmelden
				IFmnParam.Out.Edit.wStatus := MAX(59999,DINT_TO_UINT(_PmIntern.Status.diMsgAttr1));

				// Statemachine Backup zurücksetzen
				_PmIntern.enCycBackup := cs_BacIdle;
				// Kommando muss zurückgenommen werden
				_PmIntern.enCycIfState := cs_IfReady;

				_LogEntryIn.wErrorNo := _MNPARAM_LOG_ENDBACKUP_FAILED;
				_LogEntryIn.lAttr1 := IFmnParam.Out.Edit.wStatus;
				_InsertRB(wPtrStart := _wPtrRBstart, wPtrRead := _wPtrRBread, wPtrWrite := _wPtrRBwrite);

			END_IF

		cs_IfRestore:

			// Warten bis Import/Restore fertig ist
			IF _PmIntern.enCycImpState = cs_ImpRdySuccess THEN

				// ERFOLGE

				// Rückmeldung
				IFmnParam.Out.Edit.wStatus := MNPARAM_STAT_RESTORE_OK;

				// Statemachine Import zurücksetzen
				_PmIntern.enCycImpState := cs_ImpIdle;
				// Kommando muss zurückgenommen werden
				_PmIntern.enCycIfState := cs_IfReady;

				_LogEntryIn.wErrorNo := _MNPARAM_LOG_ENDRESTORE_SUCC;
				_InsertRB(wPtrStart := _wPtrRBstart, wPtrRead := _wPtrRBread, wPtrWrite := _wPtrRBwrite);

				_actFillNamelist;

			ELSIF _PmIntern.enCycImpState = cs_ImpRdyFault THEN

				// FEHLER

				// Status zurückmelden
				IFmnParam.Out.Edit.wStatus := MAX(59999,DINT_TO_UINT(_PmIntern.Status.diMsgAttr1));

				// Statemachine Import zurücksetzen
				_PmIntern.enCycImpState := cs_ImpIdle;
				// Kommando muss zurückgenommen werden
				_PmIntern.enCycIfState := cs_IfReady;

				_LogEntryIn.wErrorNo := _MNPARAM_LOG_ENDRESTORE_FAILED;
				_LogEntryIn.lAttr1 := IFmnParam.Out.Edit.wStatus;
				_InsertRB(wPtrStart := _wPtrRBstart, wPtrRead := _wPtrRBread, wPtrWrite := _wPtrRBwrite);

			END_IF

		cs_IfReady:

			// Warten, bis das Kommando zurückgenommen wurde. Bei Warnung mindestzeit abwarten
			IF IFmnParam.In.Edit.wCommand = MNPARAM_CMD_NOCOMMAND AND (_PmIntern.Status.wMsgNumber = 0 OR TONwarn2.Q) THEN

				// Rückmeldung
				IFmnParam.Out.Edit.wStatus := MNPARAM_STAT_NOCOMMAND;

				// Meldung zurücksetzen
				brsmemset(ADR(_PmIntern.Status), 0, SIZEOF(_PmIntern.Status));
				_PmIntern.Status.wFunction_ID := MNPARAM_FUNCTIONID;

				// Interface zur Applikation wieder bereit schalten
				_PmIntern.enCycIfState := cs_IfIdle;

			END_IF

	END_CASE

	// Warnung soll mindestens 4 Sekunden anstehen
	TONwarn2(IN := _PmIntern.enCycIfState = cs_IfReady, PT := T#4s);

END_ACTION
```

#### _actFillEditNum.st
```iecst
(********************************************************************
 * COPYRIGHT -- Herbert Kannegiesser GmbH
 ********************************************************************
 * Program: mnParam
 * File: _actFillEditNum.st
 * Author: hunholz
 * Created: March 21, 2012
 ********************************************************************
 * Implementation of program mnParam
 ********************************************************************)

(* Attribute und Werte füllen *)
ACTION _actFillEditNum:

	// Attribute übertragen

	IFmnParam.Out.Edit.AttrNum[_wActRow].wType := _pDoParamNum.ParamNum[_wActRefIdx].bRowType + MNPARAM_CSV_DAT_NUM;
	IFmnParam.Out.Edit.AttrNum[_wActRow].wUnit := _pDoParamNum.ParamNum[_wActRefIdx].wUnitID;
	IFmnParam.Out.Edit.AttrNum[_wActRow].wFunctionID := _pDoParamNum.ParamNum[_wActRefIdx].wFunction_ID;
	IFmnParam.Out.Edit.AttrNum[_wActRow].wParamNo := _pDoParamNum.ParamNum[_wActRefIdx].wParNo;
	IFmnParam.Out.Edit.AttrNum[_wActRow].wParIdx := _wActRefIdx;
	IFmnParam.Out.Edit.AttrNum[_wActRow].wArrIdx[1] := _pDoContainerNum.CsvNum[_wActIdx].wArrIdx1;
	IFmnParam.Out.Edit.AttrNum[_wActRow].wArrIdx[2] := _pDoContainerNum.CsvNum[_wActIdx].wArrIdx2;
	IFmnParam.Out.Edit.AttrNum[_wActRow].wArrIdx[3] := _pDoContainerNum.CsvNum[_wActIdx].wArrIdx3;
	IFmnParam.Out.Edit.AttrNum[_wActRow].wArrIdx[4] := _pDoContainerNum.CsvNum[_wActIdx].wArrIdx4;

	_pDigits := ADR(IFmnParam.Out.Edit.AttrNum[_wActRow].lDigits);
	_pUnit := ADR(IFmnParam.Out.Edit.AttrNum[_wActRow].sUnit);

	IF _pDoParamNum.ParamNum[_wActRefIdx].bRowType = 0 THEN

		// INT
		IFmnParam.Out.Edit.AttrNum[_wActRow].rDefault := kgUnitconfREALtoDisplay(DINT_TO_REAL(_pDoParamNum.ParamNum[_wActRefIdx].diDefValue),_pDoParamNum.ParamNum[_wActRefIdx].wUnitID,IFmnParam.In.Edit.bLocUnit, _pDigits, _pUnit);
		IFmnParam.Out.Edit.AttrNum[_wActRow].rMax := kgUnitconfREALtoDisplay(DINT_TO_REAL(_pDoParamNum.ParamNum[_wActRefIdx].diMaxValue),_pDoParamNum.ParamNum[_wActRefIdx].wUnitID,IFmnParam.In.Edit.bLocUnit, 0, 0);
		IFmnParam.Out.Edit.AttrNum[_wActRow].rMin := kgUnitconfREALtoDisplay(DINT_TO_REAL(_pDoParamNum.ParamNum[_wActRefIdx].diMinValue),_pDoParamNum.ParamNum[_wActRefIdx].wUnitID,IFmnParam.In.Edit.bLocUnit, 0, 0);

	ELSE

		// REAL
		_prValue ACCESS ADR(_pDoParamNum.ParamNum[_wActRefIdx].diDefValue);
		IFmnParam.Out.Edit.AttrNum[_wActRow].rDefault := kgUnitconfREALtoDisplay(_prValue,_pDoParamNum.ParamNum[_wActRefIdx].wUnitID,IFmnParam.In.Edit.bLocUnit, _pDigits, _pUnit);
		_prValue ACCESS ADR(_pDoParamNum.ParamNum[_wActRefIdx].diMaxValue);
		IFmnParam.Out.Edit.AttrNum[_wActRow].rMax := kgUnitconfREALtoDisplay(_prValue,_pDoParamNum.ParamNum[_wActRefIdx].wUnitID,IFmnParam.In.Edit.bLocUnit, 0, 0);
		_prValue ACCESS ADR(_pDoParamNum.ParamNum[_wActRefIdx].diMinValue);
		IFmnParam.Out.Edit.AttrNum[_wActRow].rMin := kgUnitconfREALtoDisplay(_prValue,_pDoParamNum.ParamNum[_wActRefIdx].wUnitID,IFmnParam.In.Edit.bLocUnit, 0, 0);

	END_IF

	// Wert übergeben

	IF _pDoParamNum.ParamNum[_wActRefIdx].bRowType = 0 THEN
		_EditNumValues.rVal[_wActRow] := kgUnitconfREALtoDisplay(DINT_TO_REAL(_pDoContainerNum.CsvNum[_wActIdx].diValue),_pDoParamNum.ParamNum[_wActRefIdx].wUnitID,IFmnParam.In.Edit.bLocUnit, 0, 0);
	ELSE
		_prValue ACCESS ADR(_pDoContainerNum.CsvNum[_wActIdx].diValue);
		_EditNumValues.rVal[_wActRow] := kgUnitconfREALtoDisplay(_prValue,_pDoParamNum.ParamNum[_wActRefIdx].wUnitID,IFmnParam.In.Edit.bLocUnit, 0, 0);
	END_IF

	_EditNumValues.wIdx[_wActRow] := _wActIdx;

	// Texte übergeben (Binäre Suche)

	IF IFmnTxt.Out.wSelectLanguageStatus = ERR_OK AND IFmnTxt.Out.ptrFunctionTxtList <> 0 AND IFmnTxt.Out.ptrInstanceTxtList <> 0 AND
		IFmnTxt.Out.ptrParamTxtList <> 0 AND IFmnTxt.Out.ptrParamHelpTxtList <> 0 THEN

		_wIdxFunctionTxt := _BinSearchTxtLine(IFmnParam.Out.Edit.AttrNum[_wActRow].wFunctionID, 0, IFmnTxt.Out.ptrFunctionTxtList, IFmnTxt.Out.wCntFunctionTxt);

		_wIdxInstanceTxt := _BinSearchTxtLine(IFmnParam.Out.Edit.AttrNum[_wActRow].wFunctionID, IFmnParam.Out.Edit.AttrNum[_wActRow].wArrIdx[1],
		IFmnTxt.Out.ptrInstanceTxtList, IFmnTxt.Out.wCntInstanceTxt);

		_wIdxParamTxt := _BinSearchTxtLine(IFmnParam.Out.Edit.AttrNum[_wActRow].wFunctionID, IFmnParam.Out.Edit.AttrNum[_wActRow].wParamNo,
		IFmnTxt.Out.ptrParamTxtList, IFmnTxt.Out.wCntParamTxt);

		_wIdxParamHlpTxt := _BinSearchHlpTxtLine(IFmnParam.Out.Edit.AttrNum[_wActRow].wFunctionID, IFmnParam.Out.Edit.AttrNum[_wActRow].wParamNo,
		IFmnTxt.Out.ptrParamHelpTxtList, IFmnTxt.Out.wCntParamHlpTxt);

		IFmnParam.Out.Edit.AttrNum[_wActRow].utfParameterName := "";
		IFmnParam.Out.Edit.AttrNum[_wActRow].utfParameterHelpTxt := "";
		IFmnParam.Out.Edit.AttrNum[_wActRow].utfFunction := "";
		IFmnParam.Out.Edit.AttrNum[_wActRow].utfInstance := "";
		_wLenUtf := 0;

		IF _wIdxFunctionTxt <> 65535 THEN
			_pFunctionTxt ACCESS IFmnTxt.Out.ptrFunctionTxtList;
			brwcsncat(ADR(IFmnParam.Out.Edit.AttrNum[_wActRow].utfFunction), ADR(_pFunctionTxt[_wIdxFunctionTxt].utfText), 31);
			IF NOT MNPARAM_DISABLE_FILLEDIT_FUNCT THEN
				brwcsncat(ADR(IFmnParam.Out.Edit.AttrNum[_wActRow].utfParameterName), ADR(IFmnParam.Out.Edit.AttrNum[_wActRow].utfFunction), 63-_wLenUtf);
				_wLenUtf := UDINT_TO_UINT(brwcslen(ADR(IFmnParam.Out.Edit.AttrNum[_wActRow].utfParameterName)));
				brwcsncat(ADR(IFmnParam.Out.Edit.AttrNum[_wActRow].utfParameterName), ADR("."), 63-_wLenUtf);
				_wLenUtf := UDINT_TO_UINT(brwcslen(ADR(IFmnParam.Out.Edit.AttrNum[_wActRow].utfParameterName)));
			END_IF
		END_IF

		IF _wIdxInstanceTxt <> 65535 THEN
			_pInstanceTxt ACCESS IFmnTxt.Out.ptrInstanceTxtList;
			brwcsncat(ADR(IFmnParam.Out.Edit.AttrNum[_wActRow].utfInstance), ADR(_pInstanceTxt[_wIdxInstanceTxt].utfText), 31);
			IF NOT MNPARAM_DISABLE_FILLEDIT_INST THEN
				brwcsncat(ADR(IFmnParam.Out.Edit.AttrNum[_wActRow].utfParameterName), ADR(IFmnParam.Out.Edit.AttrNum[_wActRow].utfInstance), 63-_wLenUtf);
				_wLenUtf := UDINT_TO_UINT(brwcslen(ADR(IFmnParam.Out.Edit.AttrNum[_wActRow].utfParameterName)));
				brwcsncat(ADR(IFmnParam.Out.Edit.AttrNum[_wActRow].utfParameterName), ADR("."), 63-_wLenUtf);
				_wLenUtf := UDINT_TO_UINT(brwcslen(ADR(IFmnParam.Out.Edit.AttrNum[_wActRow].utfParameterName)));
			END_IF
		END_IF

		IF _wIdxParamTxt <> 65535 THEN
			_pParamTxt ACCESS IFmnTxt.Out.ptrParamTxtList;
			brwcsncat(ADR(IFmnParam.Out.Edit.AttrNum[_wActRow].utfParameterName), ADR(_pParamTxt[_wIdxParamTxt].utfText), 63-_wLenUtf);
		END_IF

		IF _wIdxParamHlpTxt <> 65535 THEN
			_pParamHlpTxt ACCESS IFmnTxt.Out.ptrParamHelpTxtList;
			brwcsncat(ADR(IFmnParam.Out.Edit.AttrNum[_wActRow].utfParameterHelpTxt), ADR(_pParamHlpTxt[_wIdxParamHlpTxt].utfText), 255);
		END_IF

	END_IF

END_ACTION
```

#### _actFillEditStr.st
```iecst
(********************************************************************
 * COPYRIGHT -- Herbert Kannegiesser GmbH
 ********************************************************************
 * Program: mnParam
 * File: _actFillEditStr.st
 * Author: hunholz
 * Created: March 21, 2012
 ********************************************************************
 * Implementation of program mnParam
 ********************************************************************)

(* Attribute und Werte *)
ACTION _actFillEditStr:

	// Attribute übertragen

	IFmnParam.Out.Edit.AttrStr[_wActRow].wType := 20;
	IFmnParam.Out.Edit.AttrStr[_wActRow].wFunctionID := _pDoParamString.ParamString[_wActRefIdx].wFunction_ID;
	IFmnParam.Out.Edit.AttrStr[_wActRow].wParamNo := _pDoParamString.ParamString[_wActRefIdx].wParNo;
	IFmnParam.Out.Edit.AttrStr[_wActRow].wParIdx := _wActRefIdx;
	IFmnParam.Out.Edit.AttrStr[_wActRow].wArrIdx[1] := _pDoContainerString.CsvString[_wActIdx].wArrIdx1;
	IFmnParam.Out.Edit.AttrStr[_wActRow].wArrIdx[2] := _pDoContainerString.CsvString[_wActIdx].wArrIdx2;
	IFmnParam.Out.Edit.AttrStr[_wActRow].wArrIdx[3] := _pDoContainerString.CsvString[_wActIdx].wArrIdx3;
	IFmnParam.Out.Edit.AttrStr[_wActRow].wArrIdx[4] := _pDoContainerString.CsvString[_wActIdx].wArrIdx4;

	IFmnParam.Out.Edit.AttrStr[_wActRow].utfDefault := _pDoParamString.ParamString[_wActRefIdx].utfDefValue;
	IFmnParam.Out.Edit.AttrStr[_wActRow].wMaxLength := _pDoParamString.ParamString[_wActRefIdx].bLenght;

	// Wert übergeben

	_EditStrValues.utfVal[_wActRow] := _pDoContainerString.CsvString[_wActIdx].utfValue;
	_EditStrValues.xSave[_wActRow] := FALSE;
	_EditStrValues.wIdx[_wActRow] := _wActIdx;

	// Texte übergeben (Binäre Suche)

	IF IFmnTxt.Out.wSelectLanguageStatus = ERR_OK AND IFmnTxt.Out.ptrFunctionTxtList <> 0 AND IFmnTxt.Out.ptrInstanceTxtList <> 0 AND
		IFmnTxt.Out.ptrParamTxtList <> 0 AND IFmnTxt.Out.ptrParamHelpTxtList <> 0 THEN

		_wIdxFunctionTxt := _BinSearchTxtLine(IFmnParam.Out.Edit.AttrStr[_wActRow].wFunctionID, 0, IFmnTxt.Out.ptrFunctionTxtList, IFmnTxt.Out.wCntFunctionTxt);

		_wIdxInstanceTxt := _BinSearchTxtLine(IFmnParam.Out.Edit.AttrStr[_wActRow].wFunctionID, IFmnParam.Out.Edit.AttrStr[_wActRow].wArrIdx[1],
		IFmnTxt.Out.ptrInstanceTxtList, IFmnTxt.Out.wCntInstanceTxt);

		_wIdxParamTxt := _BinSearchTxtLine(IFmnParam.Out.Edit.AttrStr[_wActRow].wFunctionID, IFmnParam.Out.Edit.AttrStr[_wActRow].wParamNo,
		IFmnTxt.Out.ptrParamTxtList, IFmnTxt.Out.wCntParamTxt);

		_wIdxParamHlpTxt := _BinSearchHlpTxtLine(IFmnParam.Out.Edit.AttrStr[_wActRow].wFunctionID, IFmnParam.Out.Edit.AttrStr[_wActRow].wParamNo,
		IFmnTxt.Out.ptrParamHelpTxtList, IFmnTxt.Out.wCntParamHlpTxt);

		IFmnParam.Out.Edit.AttrStr[_wActRow].utfParameterName := "";
		IFmnParam.Out.Edit.AttrStr[_wActRow].utfParameterHelpTxt := "";
		IFmnParam.Out.Edit.AttrStr[_wActRow].utfFunction := "";
		IFmnParam.Out.Edit.AttrStr[_wActRow].utfInstance := "";
		_wLenUtf := 0;

		IF _wIdxFunctionTxt <> 65535 THEN
			_pFunctionTxt ACCESS IFmnTxt.Out.ptrFunctionTxtList;
			brwcsncat(ADR(IFmnParam.Out.Edit.AttrStr[_wActRow].utfFunction), ADR(_pFunctionTxt[_wIdxFunctionTxt].utfText), 31);
			IF NOT MNPARAM_DISABLE_FILLEDIT_FUNCT THEN
				brwcsncat(ADR(IFmnParam.Out.Edit.AttrStr[_wActRow].utfParameterName), ADR(IFmnParam.Out.Edit.AttrStr[_wActRow].utfFunction), 63-_wLenUtf);
				_wLenUtf := UDINT_TO_UINT(brwcslen(ADR(IFmnParam.Out.Edit.AttrStr[_wActRow].utfParameterName)));
				brwcsncat(ADR(IFmnParam.Out.Edit.AttrStr[_wActRow].utfParameterName), ADR("."), 63-_wLenUtf);
				_wLenUtf := UDINT_TO_UINT(brwcslen(ADR(IFmnParam.Out.Edit.AttrStr[_wActRow].utfParameterName)));
			END_IF
		END_IF

		IF _wIdxInstanceTxt <> 65535 THEN
			_pInstanceTxt ACCESS IFmnTxt.Out.ptrInstanceTxtList;
			brwcsncat(ADR(IFmnParam.Out.Edit.AttrStr[_wActRow].utfInstance), ADR(_pInstanceTxt[_wIdxInstanceTxt].utfText), 31);
			IF NOT MNPARAM_DISABLE_FILLEDIT_INST THEN
				brwcsncat(ADR(IFmnParam.Out.Edit.AttrStr[_wActRow].utfParameterName), ADR(IFmnParam.Out.Edit.AttrStr[_wActRow].utfInstance), 63-_wLenUtf);
				_wLenUtf := UDINT_TO_UINT(brwcslen(ADR(IFmnParam.Out.Edit.AttrStr[_wActRow].utfParameterName)));
				brwcsncat(ADR(IFmnParam.Out.Edit.AttrStr[_wActRow].utfParameterName), ADR("."), 63-_wLenUtf);
				_wLenUtf := UDINT_TO_UINT(brwcslen(ADR(IFmnParam.Out.Edit.AttrStr[_wActRow].utfParameterName)));
			END_IF
		END_IF

		IF _wIdxParamTxt <> 65535 THEN
			_pParamTxt ACCESS IFmnTxt.Out.ptrParamTxtList;
			brwcsncat(ADR(IFmnParam.Out.Edit.AttrStr[_wActRow].utfParameterName), ADR(_pParamTxt[_wIdxParamTxt].utfText), 63-_wLenUtf);
		END_IF

		IF _wIdxParamHlpTxt <> 65535 THEN
			_pParamHlpTxt ACCESS IFmnTxt.Out.ptrParamHelpTxtList;
			brwcsncat(ADR(IFmnParam.Out.Edit.AttrStr[_wActRow].utfParameterHelpTxt), ADR(_pParamHlpTxt[_wIdxParamHlpTxt].utfText), 255);
		END_IF

	END_IF

END_ACTION
```

#### _actFillNamelist.st
```iecst
(********************************************************************
 * COPYRIGHT -- Herbert Kannegiesser GmbH
 ********************************************************************
 * Program: mnParam
 * File: _actFillNamelist.st
 * Author: hunholz
 * Created: March 30, 2012
 ********************************************************************
 * Implementation of program mnParam
 ********************************************************************)

(* Namensliste für Programme füllen *)
ACTION _actFillNamelist:

	IFmnParam.Out.Edit.wCntNamelist := 0;
	brsmemset(ADR(IFmnParam.Out.Edit.wNameListNo), 0, SIZEOF(IFmnParam.Out.Edit.wNameListNo));
	brsmemset(ADR(IFmnParam.Out.Edit.utfNameListName), 0, SIZEOF(IFmnParam.Out.Edit.utfNameListName));

	IF IFmnParam.Out.Edit.wIdxContainerNamelist <= MNPARAM_MAXIDX_CONTAINER THEN

		IF _pDoContainer.Container[IFmnParam.Out.Edit.wIdxContainerNamelist].bDirectParam = 0 AND _pDoContainer.Container[IFmnParam.Out.Edit.wIdxContainerNamelist].wDimension > 0 THEN

			_wActListIdx := 1;

			FOR _k := 0 TO _pDoContainer.Container[IFmnParam.Out.Edit.wIdxContainerNamelist].wDimension-1 DO

				IF _PmIntern.TOC.TocEntry[_PmIntern.TOC.wStartIdx[IFmnParam.Out.Edit.wIdxContainerNamelist] + _k].xExist THEN

					IFmnParam.Out.Edit.wNameListNo[_wActListIdx] := _pDoContainer.Container[IFmnParam.Out.Edit.wIdxContainerNamelist].wMinBound + _k;

					_DefineActContainer(Enable := TRUE, bContainerIdx := UINT_TO_USINT(IFmnParam.Out.Edit.wIdxContainerNamelist), wInstanceIdx := IFmnParam.Out.Edit.wNameListNo[_wActListIdx], pIntern := ADR(_PmIntern));

					IF _DefineActContainer.Status = ERR_OK THEN

						IF IFmnParam.Out.Edit.wParIdxNamelist > 0 AND IFmnParam.Out.Edit.wParIdxNamelist <= _PmIntern.DataObjects.MaxIndex.lParamString THEN

							_diProgname(enable := TRUE, pName := ADR(_PmIntern.ActContainer.sDoNameString));

							IF _diProgname.status = ERR_OK THEN

								IFmnParam.Out.Edit.utfNameListName[_wActListIdx] := UINT_TO_WSTRING(_k);
								brwcscat(ADR(IFmnParam.Out.Edit.utfNameListName[_wActListIdx]), ADR(" - "));

								// Datenobjekt mit aktuellen String Parametern wurde gefunden
								_PmIntern.CSVDataObjects.Adress.lCSVString := _diCSVString.pDatObjMem;
								_PmIntern.CSVDataObjects.Size.lCSVString := _diCSVString.len;
								_PmIntern.CSVDataObjects.Idents.lCSVString := _diCSVString.ident;

								_pDoProgContainer ACCESS _diProgname.pDatObjMem;
								_lMaxIndexProgContainer := ( (_pDoProgContainer.Header.Do.lActEndPos - SIZEOF(mnParam_CsvDynHeader_typ)) / SIZEOF(_pDoProgContainer.CsvString[1]) );

								// Suche Parameter-Containerindex anhand des Parameterindex und der 4 möglichen Array-Werte
								_binarySearchString.enable := TRUE;
								_binarySearchString.CsvStructString.wIdxStringPar 	:= IFmnParam.Out.Edit.wParIdxNamelist;
								_binarySearchString.CsvStructString.wArrIdx1 		:= 0;
								_binarySearchString.CsvStructString.wArrIdx2 		:= 0;
								_binarySearchString.CsvStructString.wArrIdx3 		:= 0;
								_binarySearchString.CsvStructString.wArrIdx4 		:= 0;
								_binarySearchString.lpList 							:=  _diProgname.pDatObjMem;
								_binarySearchString.lMaxRow 						:= _lMaxIndexProgContainer;

								_binarySearchString();

								// Wurde der Parameter im Container gefunden ?
								IF _binarySearchString.status = ERR_OK THEN

									brwcscat(ADR(IFmnParam.Out.Edit.utfNameListName[_wActListIdx]), ADR(_pDoProgContainer.CsvString[_binarySearchString.lFoundRow].utfValue));

								END_IF

							END_IF

						END_IF

						IFmnParam.Out.Edit.wCntNamelist := _wActListIdx;
						_wActListIdx := _wActListIdx + 1;

						IF _wActListIdx > MNPARAM_CNT_NAMELIST THEN
							// Abbrechen, wenn die Liste voll ist
							EXIT;
						END_IF

					ELSE

						IFmnParam.Out.Edit.wNameListNo[_wActListIdx] := 0;

					END_IF

				END_IF

			END_FOR

		END_IF

	END_IF

END_ACTION
```

#### _actImpModel.st
```iecst
(********************************************************************
 * COPYRIGHT -- Herbert Kannegiesser GmbH
 ********************************************************************
 * Program: mnParam
 * File: _actImpModel.st
 * Author: hunholz
 * Created: June 04, 2012
 ********************************************************************
 * Implementation of program mnParam
 ********************************************************************)

(* Datenmodell von USB-Stick importieren *)
ACTION _actImpModel:

	CASE _wStateImportDatamodel OF

		0:	// USB Device erstellen
			_sDevString := CONCAT('/DEVICE=',IFmnSystem.Out.sInterfaceUSB);
			_DevLink(enable := TRUE, pDevice := ADR(_MNPARAM_TEMP_USBDEV), pParam := ADR(_sDevString));

			IF _DevLink.status = ERR_OK THEN

				_sImportDevice := _MNPARAM_TEMP_USBDEV;
				_lDevLinkHandle := _DevLink.handle;

				_wStateImportDatamodel := 10;

			ELSIF _DevLink.status <> ERR_FUB_BUSY THEN

				_xModelImportChecked := TRUE;
				_xParamOK := NOT _xSysError;

			END_IF

		10:	// Nach dem Pfad SetupKG suchen

			_DirInfo(enable := TRUE, pDevice := ADR(_sImportDevice), pPath := ADR(MNPARAM_PATH_IMPORTDATAMODEL));

			IF _DirInfo.status = ERR_OK THEN

				_xFoundDM := FALSE;
				_lDirNum := _DirInfo.dirnum;

				IF _xRBReady THEN
					_LogEntryIn.wErrorNo := _MNPARAM_LOG_FOUNDIMPDIR;
					_LogEntryIn.lAttr1 := _lDirNum;
					_InsertRB(wPtrStart := _wPtrRBstart, wPtrRead := _wPtrRBread, wPtrWrite := _wPtrRBwrite);
				END_IF

				IF _lDirNum = 0 THEN

					_wStateImportDatamodel := 999;

				ELSE

					_wStateImportDatamodel := 20;

				END_IF

			ELSIF _DirInfo.status <> ERR_FUB_BUSY THEN

				_wStateImportDatamodel := 999;

			END_IF

		20:		// Search for DataModel.csv

			_sTestFile := CONCAT(MNPARAM_PATH_IMPORTDATAMODEL,'\PM\DataModel.csv');

			_FileInfo(enable := TRUE, pDevice := ADR(_sImportDevice), pName := ADR(_sTestFile), pInfo := ADR(_fiDataModel));

			IF _FileInfo.status <> ERR_FUB_BUSY THEN

				_xFoundDM := _FileInfo.status = ERR_OK;

				IF _xFoundDM THEN

					_wStateImportDatamodel := 40;

				ELSE

					_wStateImportDatamodel := 30;

				END_IF

			END_IF

		30:		// Search for _mnr.csv

			_sTestFile := CONCAT(MNPARAM_PATH_IMPORTDATAMODEL,'\PM\_mnr.csv');

			_FileInfo(enable := TRUE, pDevice := ADR(_sImportDevice), pName := ADR(_sTestFile), pInfo := ADR(_fiMNR));

			IF _FileInfo.status <> ERR_FUB_BUSY THEN

				_xFoundDM := _FileInfo.status = ERR_OK;

				_wStateImportDatamodel := 40;

			END_IF

		40:		// Copy all

			_DirCopy(enable := TRUE, pSrcDev := ADR(_sImportDevice), pSrcDir := ADR(MNPARAM_PATH_IMPORTDATAMODEL), pDestDev := ADR(KG_DEVICE_COMPACTFLASH), pDestDir := ADR(''), option := fiOVERWRITE + fiRECURSIVE);

			IF _DirCopy.status <> ERR_FUB_BUSY THEN

				_xImpDMOK := _DirCopy.status = ERR_OK;

				_wStateImportDatamodel := 999;

			END_IF

		999:	// Device unlinken

			_DevUnlink(enable := TRUE, handle := _lDevLinkHandle);

			IF _DevUnlink.status <> ERR_FUB_BUSY THEN

				_wStateImportDatamodel := 65535;

				_xModelImportChecked := TRUE;

				IF NOT _xFoundDM AND _xImpDMOK THEN

					_xParamOK := NOT _xSysError;

				END_IF

			END_IF

	END_CASE

END_ACTION
```

### Library Logical/Standard/Kanlink/KGFramework/Pkg_mnParam/mnParamLib (IEC)
Depends on: astime

#### mnParamLib.typ - Exported data types
```iecst
(********************************************************************
 * COPYRIGHT -- Microsoft
 ********************************************************************
 * Library: mnParamLib
 * File: mnParamLib.typ
 * Author: Reese_Markus
 * Created: July 25, 2011
 ********************************************************************
 * Data types of library mnParamLib
 ********************************************************************)
(**** Zeilen Strukturen ****)

TYPE
	mnParam_HeaderDoRow_typ : 	STRUCT
		lActEndPos : UDINT;
	END_STRUCT;
	mnParam_HeaderVersionRow_typ : 	STRUCT
		wVersion : UINT; (*Versionsnummer des Datenmodells*)
		wReserve : UINT;
		dtTimestamp : DATE_AND_TIME; (*Speicherdatum der Datei*)
		utfMachineType : WSTRING[11]; (*Maschinentyp*)
		utfMachineSubType : WSTRING[11]; (*MaschinenSubTyp*)
	END_STRUCT;
	mnParam_HeaderTimeRow_typ : 	STRUCT
		dtTimestamp : DATE_AND_TIME; (*Zeitstempel der Datei*)
	END_STRUCT;
	mnParam_HeaderMachineNoRow_typ : 	STRUCT
		utfMachineNo : WSTRING[15]; (*Maschinennummer*)
	END_STRUCT;
	mnParam_ContainerHeader_typ : 	STRUCT
		xWriteProtected : BOOL; (*Wird gesetzt, wenn Datencontainer im PM-Verzeichnis liegt*)
		bReserve : ARRAY[0..2]OF USINT;
	END_STRUCT;
	mnParam_CProw_typ : 	STRUCT
		sCategory : STRING[11];
		utfCategoryName : WSTRING[31];
		dtTimeStamp : DATE_AND_TIME;
		wProgramNo : UINT;
		wLoadrate : UINT;
		rSoilfactor : REAL;
		wColFor : UINT;
		wColBack : UINT;
	END_STRUCT;
	mnParam_LCIDrow_typ : 	STRUCT
		LCID : UINT;
		utfName : WSTRING[31];
	END_STRUCT;
	mnParam_HelpTxtRow_typ : 	STRUCT
		LCID : UINT;
		FunctionID : UINT;
		TextNo : UINT;
		utfHelpText : WSTRING[255];
	END_STRUCT;
	mnParam_TxtRow_typ : 	STRUCT
		LCID : UINT;
		FunctionID : UINT;
		TextNo : UINT;
		utfText : WSTRING[63];
	END_STRUCT;
	mnParam_ContainerRow_typ : 	STRUCT
		siContainerID : SINT; (*<0, 0 ist für _ConfigPar reserviert*)
		bDirectParam : USINT; (*0 - indirekt, 1 - direkt*)
		sNameDataObj : STRING[11]; (*Name des Daten-Objekts*)
		sNameCsv : STRING[31]; (*Name der CSV-Datei*)
		wMinBound : UINT; (*Kleinster Index, wenn es mehrere Container gibt, Dimension muss dazu größer 0 sein*)
		wDimension : UINT; (*0 - Es gibt nur einen Container, >0 - Anzahl der Container, aufsteigend nummeriert*)
		sStrucRoot : STRING[31]; (*Name des Wurzelelements*)
		lCountNum : DINT;
		lCountString : DINT;
	END_STRUCT;
	mnParam_LogicalStructRow_typ : 	STRUCT
		wLogStrucNo : UINT; (*Eindeutiger Idex für das logische Strukturelement, >0*)
		wMinBound : UINT; (*kleinster Index*)
		wDimension : UINT; (*0 - kein Array*)
		siWriteAccess : SINT; (*Notwendiger Benutzerlevel, um Schreibrecht für alle Parameter unterhalb dieses Knotens zu erlangen, <0 - Recht ist vererbt*)
		siVisibleAccess : SINT; (*Notwendiger Benutzerlevel, um Leserecht für alle Parameter unterhalb dieses Knotens zu erlangen.*)
		iReferenz : INT; (*<=0 - Strukturelement ist Wurzel, >0 - Strukturelement ist Kind von IdxLogStruc*)
		wRefVisible : UINT; (*Verweis auf Parameter, die die Sichtbarkeit steuern*)
		wRefText : UINT; (*Verweis auf ein Textparameter, der das Element beschriftet. Sonst wird der Text aus der Rextresource verwendet*)
		bFormatArray : USINT;
		bReserve : USINT;
		utfMachineSubType : WSTRING[11];
		utfLogStrucName : WSTRING[31];
	END_STRUCT;
	mnParam_ParamNumRow_typ : 	STRUCT
		wIdxNumPar : UINT; (*Eindeutiger Index für den Numerischen Parameter (Referenziert den Eintrag im Array auf der SPS)*)
		wFunction_ID : UINT; (*Nummer der Funktionsgruppe, zu dem der Parameter gehört*)
		wParNo : UINT; (*Eindeutige Paremeternummer innerhalb der Funktionsgruppe*)
		siWriteAccess : SINT; (*<0 - Recht ist vererbt, Notwendiger Benutzerlevel, um Schreibrecht für alle Parameter unterhalb dieses Knotens zu erlangen.*)
		siVisibleAccess : SINT; (*Notwendiger Benutzerlevel, um Leserecht für alle Parameter unterhalb dieses Knotens zu erlangen*)
		sAdresse : STRING[63]; (*Adress-String (bis zu 4 verschachtelte Arrays sind möglich)*)
		wUnitID : UINT; (*Einheitenklasse*)
		wMinBound : UINT; (*<0 - wird nicht für letzte Arraystufe herangezogen*)
		wDimension : UINT; (*0 - wird nicht für letzte Arraystufe herangezogen*)
		wReferenz : UINT; (*Verweis auf IdxLogStruc*)
		diMinValue : DINT; (*Untere Begrenzung*)
		diMaxValue : DINT; (*Obere Begrenzung*)
		diDefValue : DINT; (*Default Wert*)
		utfMachineSubType : WSTRING[11];
		wITIdx : UINT;
		bRowType : USINT; (*0 - Integer, 1 - Fließkomma*)
		bInputType : USINT;
		wRefVisible : UINT; (*Verweist auf Idx eines numerischen Parameters, der die Sichtbarkeit steuert*)
		wRefVisibleType : UINT; (*Gibt die Regel an, wie die Sichtbarkeit gesteuert wird*)
		wRefText : UINT; (*Verweist auf den Idx eines String Parameters, der in den Parameternamen eingefügt wird.*)
	END_STRUCT;
	mnParam_ParamStringRow_typ : 	STRUCT
		wIdxStringPar : UINT; (*Eindeutiger Index für den Zeichen Parameter (Referenziert den Eintrag im Array auf der SPS)*)
		wFunction_ID : UINT; (*Nummer der Funktionsgruppe, zu dem der Parameter gehört*)
		wParNo : UINT; (*Eindeutige Parameternummer innerhalb der Funktionsgruppe*)
		bLenght : USINT; (*Maximale Eingabelänge für String (max. 31 Zeichen)*)
		siWriteAccess : SINT; (*<0 - Recht ist vererbt, Notwendiger Benutzerlevel, um Schreibrecht für alle Parameter unterhalb dieses Knotens zu erlangen*)
		siVisibleAccess : SINT; (*Notwendiger Benutzlevel, um Leserecht für alle Parameter unterhalb dieses Knotens zu erlangen*)
		bReserve : USINT;
		sAdresse : STRING[63]; (*Adress-String (bis zu 4 verschachtelete Arrays sind möglich)*)
		wMinBound : UINT; (*<0 - wird nicht für letzte Arraystufe herangezogen*)
		wDimension : UINT; (*0 - wird nicht für letzte Arraystufe herangezogen*)
		wReferenz : UINT; (*Verweis auf IdxLogStruc*)
		utfDefValue : WSTRING[31]; (*Default Wert*)
		utfMachineSubType : WSTRING[11];
		wRefVisible : UINT; (*Verweist auf Idx eines numerischen Parameters, der die Sichtbarkeit steuert*)
		wRefVisibleType : UINT; (*Gibt die Regel an, wie die Sichtbarkeit gesteuert wird*)
		wRefText : UINT; (*Verweist auf den Idx eines String Parameters, der in den Parameternamen eingefügt wird.*)
	END_STRUCT;
	mnParam_CsvNumRow_typ : 	STRUCT
		wIdxNumPar : UINT; (*Eindeutiger Index für den numerischen Parameter (Referenziert den Eintrag im Array der SPS)*)
		xChanged : BOOL;
		bRowType : USINT; (*0 - Integer, 1 - Real*)
		diValue : DINT; (*Wert des Parameters*)
		wArrIdx1 : UINT; (*1. Array Index*)
		wArrIdx2 : UINT; (*2. Array Index*)
		wArrIdx3 : UINT; (*3. Array Index*)
		wArrIdx4 : UINT; (*4. Array Index*)
		utfMachineSubType : WSTRING[11];
	END_STRUCT;
	mnParam_CsvStringRow_typ : 	STRUCT
		wIdxStringPar : UINT; (*Eindeutiger Index für den Zeichen Parameter (Referenziert den Eintrag im Array der SPS)*)
		xChanged : BOOL;
		bReserve : USINT;
		utfValue : WSTRING[31]; (*Wert des Parameters*)
		wArrIdx1 : UINT; (*1. Array Index*)
		wArrIdx2 : UINT; (*2. Array Index*)
		wArrIdx3 : UINT; (*3. Array Index*)
		wArrIdx4 : UINT; (*4. Array Index*)
		utfMachineSubType : WSTRING[11];
	END_STRUCT;
	mnParam_CsvIPRow_typ : 	STRUCT
		utfIP_Adress : WSTRING[15];
		utfGateway : WSTRING[15];
	END_STRUCT;
	mnParam_CsvContent_typ : 	STRUCT
		iContainerID : SINT; (*ContainerID 0 .. -127*)
		xExist : BOOL; (*Datei existiert*)
		wInstance : UINT; (*Instanz 0 .. 65535*)
		dtTimestamp : DATE_AND_TIME; (*Zeitstempel des Containers*)
	END_STRUCT;
END_TYPE

(**** Dynamische Strukturen ****)

TYPE
	mnParam_ContainerDynHeader_typ : 	STRUCT
		Do : mnParam_HeaderDoRow_typ; (*Header - Do*)
		Version : mnParam_HeaderVersionRow_typ; (*Header - Version*)
		Time : mnParam_HeaderTimeRow_typ; (*Header - Zeitstempel*)
	END_STRUCT;
	mnParam_ContainerDyn_typ : 	STRUCT  (*Zeilen: 20*)
		Header : mnParam_ContainerDynHeader_typ;
		Container : ARRAY[0..MNPARAM_MAXIDX_CONTAINER]OF mnParam_ContainerRow_typ;
	END_STRUCT;
	mnParam_LogicalStructDyn_typ : 	STRUCT  (*Zeilen: 50*)
		Header : mnParam_ContainerDynHeader_typ;
		LogicalStruct : ARRAY[1..MNPARAM_MAXIDX_LOGICSTRUCT]OF mnParam_LogicalStructRow_typ;
	END_STRUCT;
	mnParam_ParamNumDyn_typ : 	STRUCT  (*Zeilen: 300*)
		Header : mnParam_ContainerDynHeader_typ;
		ParamNum : ARRAY[1..MNPARAM_MAXIDX_PARAMNUM]OF mnParam_ParamNumRow_typ;
	END_STRUCT;
	mnParam_ParamStringDyn_typ : 	STRUCT  (*Zeilen: 300*)
		Header : mnParam_ContainerDynHeader_typ;
		ParamString : ARRAY[1..MNPARAM_MAXIDX_PARAMSTRING]OF mnParam_ParamStringRow_typ;
	END_STRUCT;
	mnParam_CsvDynHeader_typ : 	STRUCT
		Do : mnParam_HeaderDoRow_typ; (*Header - Do*)
		Version : mnParam_HeaderVersionRow_typ; (*Header - Version*)
		Time : mnParam_HeaderTimeRow_typ; (*Header - Zeitstempel*)
		MachineNo : mnParam_HeaderMachineNoRow_typ; (*Header - Maschinen Nummer*)
		Container : mnParam_ContainerHeader_typ; (*Header - Interne Daten*)
	END_STRUCT;
	mnParam_CsvNumDyn_typ : 	STRUCT  (*Zeilen: 5000*)
		Header : mnParam_CsvDynHeader_typ;
		CsvNum : ARRAY[1..MNPARAM_MAXIDX_CSVNUM]OF mnParam_CsvNumRow_typ;
	END_STRUCT;
	mnParam_CsvStringDyn_typ : 	STRUCT  (*Zeilen: 5000*)
		Header : mnParam_CsvDynHeader_typ; (*Header - Do*)
		CsvString : ARRAY[1..MNPARAM_MAXIDX_CSVSTRING]OF mnParam_CsvStringRow_typ;
	END_STRUCT;
END_TYPE
```

#### mnParamLib.var - Exported constants
```iecst
(********************************************************************
 * COPYRIGHT -- Microsoft
 ********************************************************************
 * Library: mnParamLib
 * File: mnParamLib.var
 * Author: Reese_Markus
 * Created: July 25, 2011
 ********************************************************************
 * Constants of library mnParamLib
 ********************************************************************)
VAR CONSTANT
	MNPARAM_MAXIDX_LOGICSTRUCT : UINT := 250;
	MNPARAM_MAXIDX_CONTAINER : UINT := 20;
	MNPARAM_MAXIDX_PARAMNUM : UINT := 500;
	MNPARAM_MAXIDX_PARAMSTRING : UINT := 200;
	MNPARAM_MAXIDX_CSVNUM : UINT := 10000;
	MNPARAM_MAXIDX_CSVSTRING : UINT := 500;
END_VAR
(*Zeilenkennungen*)
VAR CONSTANT
	MNPARAM_CSV_FILEEND : UINT := 255;
	MNPARAM_CSV_COMMENT : UINT := 254;
	MNPARAM_CSV_HEADER_VERSION : UINT := 253;
	MNPARAM_CSV_HEADER_MACHINENO : UINT := 252;
	MNPARAM_CSV_HEADER_TIMESTAMP : UINT := 251;
	MNPARAM_CSV_LANGUAGEDEF : UINT := 248;
	MNPARAM_CSV_LAN_HELPTEXT : UINT := 210;
	MNPARAM_CSV_LAN_TEXT : UINT := 200;
	MNPARAM_CSV_DEF_CONTAINER : UINT := 140;
	MNPARAM_CSV_DEF_LOGSTRUC : UINT := 130;
	MNPARAM_CSV_DEF_STRING : UINT := 120;
	MNPARAM_CSV_DEF_REAL : UINT := 111;
	MNPARAM_CSV_DEF_NUM : UINT := 110;
	MNPARAM_CSV_IP : UINT := 90;
	MNPARAM_CSV_CP : UINT := 81;
	MNPARAM_CSV_TOC : UINT := 80;
	MNPARAM_CSV_DAT_STRING : UINT := 20;
	MNPARAM_CSV_DAT_REAL : UINT := 11;
	MNPARAM_CSV_DAT_NUM : UINT := 10;
END_VAR
```

#### mnParamLib.fun - Exported functions and function blocks
```iecst
(********************************************************************
 * COPYRIGHT -- Microsoft
 ********************************************************************
 * Library: mnParamLib
 * File: mnParamLib.fun
 * Author: Reese_Markus
 * Created: July 25, 2011
 ********************************************************************
 * Functions and function blocks of library mnParamLib
 ********************************************************************)

FUNCTION_BLOCK mnParam_BinarySearchInNumeric (*TODO: Add your comment here*)
	VAR_INPUT
		enable : BOOL;
		CsvStructNum : mnParam_CsvNumRow_typ;
		lpList : UDINT;
		lMaxRow : UDINT;
	END_VAR
	VAR_OUTPUT
		status : UINT;
		lFoundRow : UDINT;
	END_VAR
	VAR
		_CsvStructNumDyn : REFERENCE TO mnParam_CsvNumDyn_typ;
		_lMin : UDINT;
		_lMax : UDINT;
		_lMid : UDINT;
	END_VAR
END_FUNCTION_BLOCK

FUNCTION_BLOCK mnParam_CountLines (*Zählt die gültigen Zeilen der Datei und gibt eine Zeilenstruktur zurück*)
	VAR_INPUT
		enable : BOOL;
		MaxLines : UINT;
		pAdresses : UDINT;
		pLens : UDINT;
		pFile : UDINT;
		FileSize : UDINT;
	END_VAR
	VAR_OUTPUT
		CntLines : UINT;
		status : UINT;
	END_VAR
	VAR
		_plAdresses : REFERENCE TO ARRAY[1..20000] OF UDINT;
		_pwLens : REFERENCE TO ARRAY[1..20000] OF UINT;
		_xNewLine : BOOL;
		_p : UDINT;
		_pChar : REFERENCE TO UINT;
		_lDif : UDINT;
	END_VAR
END_FUNCTION_BLOCK

FUNCTION_BLOCK mnParam_GetCsvDat (*Parsen einer CSV-Zeile*)
	VAR_INPUT
		enable : BOOL;
		utfCsvString : WSTRING[299];
	END_VAR
	VAR_OUTPUT
		status : UINT;
		RowType : UINT;
		HeaderVersion : mnParam_HeaderVersionRow_typ;
		HeaderMachineNo : mnParam_HeaderMachineNoRow_typ;
		HeaderTime : mnParam_HeaderTimeRow_typ;
		ContainerRow : mnParam_ContainerRow_typ;
		LogicalStructRow : mnParam_LogicalStructRow_typ;
		ParamNumRow : mnParam_ParamNumRow_typ;
		ParamStringRow : mnParam_ParamStringRow_typ;
		CsvNumRow : mnParam_CsvNumRow_typ;
		CsvStringRow : mnParam_CsvStringRow_typ;
		CsvIPRow : mnParam_CsvIPRow_typ;
		CsvLCIDrow : mnParam_LCIDrow_typ;
		CsvCProw : mnParam_CProw_typ;
		csvTextRow : mnParam_TxtRow_typ;
		csvHelpTextRow : mnParam_HelpTxtRow_typ;
	END_VAR
	VAR
		_utfRowType : WSTRING[15];
		_diRowType : DINT;
		_sRowType : STRING[15];
		_utfSubString : WSTRING[255];
		_sSubString : STRING[63];
		_diVersion : DINT;
		_atodt : mnParam_atodatetime;
		_GetNextSubstring : mnParam_GetNextSubstring;
		_pUtfCsvString : UDINT;
		_diNum : DINT;
		_utfDataObj : WSTRING[11];
		_rValue : REAL;
		_pdiValue : REFERENCE TO DINT;
	END_VAR
END_FUNCTION_BLOCK

FUNCTION_BLOCK mnParam_atodatetime (*String mit ISO-Zeitformat in DATE_AND_TIME wandeln*)
	VAR_INPUT
		pStr : UDINT;
	END_VAR
	VAR_OUTPUT
		status : UINT;
		dtTimeStamp : DATE_AND_TIME;
	END_VAR
	VAR
		_wPositionInTime : UINT;
		_DateTime : DTStructure;
		_sSubString : STRING[7];
		_sStr : STRING[23];
	END_VAR
END_FUNCTION_BLOCK

FUNCTION_BLOCK mnParam_GetNextSubstring (*TODO: Add your comment here*)
	VAR_INPUT
		enable : BOOL;
	END_VAR
	VAR_OUTPUT
		status : UINT;
		Length : UDINT;
		pUtfCsvSubstring : UDINT;
		EndOfLine : BOOL;
	END_VAR
	VAR_IN_OUT
		pUtfCsvString : UDINT;
	END_VAR
	VAR
		_lLen : UDINT;
		_lAdrTab : UDINT;
		_utfSubString : WSTRING[255];
	END_VAR
END_FUNCTION_BLOCK

FUNCTION_BLOCK mnParam_GetContainerOfParamNum (*ContainerID ermitteln und Array-Grenzen*)
	VAR_INPUT
		enable : BOOL;
		pLogicStructs : UDINT;
		wMaxIdxLogicStructs : UINT;
		pParamNum : UDINT;
	END_VAR
	VAR_OUTPUT
		wMinBound : ARRAY[1..4] OF UINT;
		wDimension : ARRAY[1..4] OF UINT;
		status : UINT;
		wCountArray : UINT;
		iContainer : INT;
	END_VAR
	VAR
		_LS : REFERENCE TO ARRAY[1..MNPARAM_MAXIDX_LOGICSTRUCT] OF mnParam_LogicalStructRow_typ;
		_PN : REFERENCE TO mnParam_ParamNumRow_typ;
		_iIdxLS : INT;
		_bMaxCycle : USINT;
		_i : UINT;
	END_VAR
END_FUNCTION_BLOCK

FUNCTION GetArrayPV : UINT (*Liefert PV-Adresse mit Indizes*)
	VAR_INPUT
		pPV : UDINT;
		pStructRoot : UDINT;
		pPVFilled : UDINT;
		idx1 : UINT;
		idx2 : UINT;
		idx3 : UINT;
		idx4 : UINT;
	END_VAR
	VAR
		_p : INT;
		_sIndex : STRING[7];
		_GetArrayPV : REFERENCE TO STRING[63];
	END_VAR
END_FUNCTION

FUNCTION_BLOCK mnParam_WritePVNum (*DINT auf beliebige, numerische Variable schreiben*)
	VAR_INPUT
		pAdress : UDINT;
		diValue : DINT;
	END_VAR
	VAR_OUTPUT
		status : UINT;
	END_VAR
	VAR
		_lPVadress : UDINT;
		_lPVlen : UDINT;
		_lPVdataType : UDINT;
		_lDataLen : UDINT;
		_wDataDimension : UINT;
		_pBool : REFERENCE TO BOOL;
		_pSint : REFERENCE TO SINT;
		_pInt : REFERENCE TO INT;
		_pDint : REFERENCE TO DINT;
		_pUsint : REFERENCE TO USINT;
		_pUint : REFERENCE TO UINT;
		_pUdint : REFERENCE TO UDINT;
		_pDT : REFERENCE TO DATE_AND_TIME;
		_pT : REFERENCE TO TIME;
		_pReal : REFERENCE TO REAL;
	END_VAR
END_FUNCTION_BLOCK

FUNCTION_BLOCK mnParam_WritePVrNum (*DINT auf beliebige, numerische Variable schreiben*)
	VAR_INPUT
		pAdress : UDINT;
		rValue : REAL;
	END_VAR
	VAR_OUTPUT
		status : UINT;
	END_VAR
	VAR
		_lPVadress : UDINT;
		_lPVlen : UDINT;
		_lPVdataType : UDINT;
		_lDataLen : UDINT;
		_wDataDimension : UINT;
		_pReal : REFERENCE TO REAL;
	END_VAR
END_FUNCTION_BLOCK

FUNCTION_BLOCK mnParam_GetContainerOfParamStrin (*Container für String-Parameter bestimmen*)
	VAR_INPUT
		enable : BOOL;
		pLogicStructs : UDINT;
		wMaxIdxLogicStructs : UINT;
		pParamString : UDINT;
	END_VAR
	VAR_OUTPUT
		status : UINT;
		wMinBound : ARRAY[1..4] OF UINT;
		wDimension : ARRAY[1..4] OF UINT;
		wCountArray : UINT;
		iContainer : INT;
	END_VAR
	VAR
		_LS : REFERENCE TO ARRAY[1..MNPARAM_MAXIDX_LOGICSTRUCT] OF mnParam_LogicalStructRow_typ;
		_PS : REFERENCE TO mnParam_ParamStringRow_typ;
		_bMaxCycle : USINT;
		_iIdxLS : INT;
		_i : UINT;
	END_VAR
END_FUNCTION_BLOCK

FUNCTION_BLOCK mnParam_WritePVString (*Schreibe String-Variable*)
	VAR_INPUT
		pAdress : UDINT;
		p_utfValue : UDINT;
	END_VAR
	VAR_OUTPUT
		status : UINT;
	END_VAR
	VAR
		_lPVadress : UDINT;
		_lPVlen : UDINT;
		_lPVdataType : UDINT;
		_lDataLen : UDINT;
		_wDataDimension : UINT;
		_utfValue : ARRAY[0..31] OF UINT;
	END_VAR
END_FUNCTION_BLOCK

FUNCTION_BLOCK mnParam_BinarySearchInString (*Binärsuche von CSV-String-Container-Zeilen*)
	VAR_INPUT
		enable : BOOL;
		lpList : UDINT;
		lMaxRow : UDINT;
		CsvStructString : mnParam_CsvStringRow_typ;
	END_VAR
	VAR_OUTPUT
		status : UINT;
		lFoundRow : UDINT;
	END_VAR
	VAR
		_CsvStructStringDyn : REFERENCE TO mnParam_CsvStringDyn_typ;
		_lMin : UDINT;
		_lMax : UDINT;
		_lMid : UDINT;
	END_VAR
END_FUNCTION_BLOCK

FUNCTION_BLOCK mnParam_WriteCSV255_Mem (*File-Ende schreiben*)
	VAR_INPUT
		enable : BOOL;
		pMem : UDINT;
		lMaxSize : UDINT;
	END_VAR
	VAR_OUTPUT
		status : UINT;
	END_VAR
	VAR_IN_OUT
		lSize : UDINT;
	END_VAR
	VAR
		_pUtfString : REFERENCE TO ARRAY[0..4] OF UINT;
	END_VAR
END_FUNCTION_BLOCK

FUNCTION_BLOCK mnParam_WriteBOM_Mem (*Byte Order Mark*)
	VAR_INPUT
		enable : BOOL;
		pMem : UDINT;
		lMaxSize : UDINT;
	END_VAR
	VAR_OUTPUT
		status : UINT;
	END_VAR
	VAR_IN_OUT
		lSize : UDINT;
	END_VAR
	VAR
		_pUtfString : REFERENCE TO UINT;
	END_VAR
END_FUNCTION_BLOCK

FUNCTION_BLOCK mnParam_WriteCSV254_Mem (*Kommentarzeile schreiben*)
	VAR_INPUT
		enable : BOOL;
		pMem : UDINT;
		lMaxSize : UDINT;
		sComment : STRING[63];
	END_VAR
	VAR_OUTPUT
		status : UINT;
	END_VAR
	VAR_IN_OUT
		lSize : UDINT;
	END_VAR
	VAR
		_pUtfString : REFERENCE TO ARRAY[0..3] OF UINT;
	END_VAR
END_FUNCTION_BLOCK

FUNCTION_BLOCK mnParam_WriteNewline_Mem (*Leerzeile*)
	VAR_INPUT
		enable : BOOL;
		pMem : UDINT;
		lMaxSize : UDINT;
	END_VAR
	VAR_OUTPUT
		status : UINT;
	END_VAR
	VAR_IN_OUT
		lSize : UDINT;
	END_VAR
	VAR
		_pUtfString : REFERENCE TO ARRAY[0..1] OF UINT;
	END_VAR
END_FUNCTION_BLOCK

FUNCTION_BLOCK mnParam_datetimetoa (*Wandelt Datum Zeit in ISO String*)
	VAR_INPUT
		dtTimestamp : DATE_AND_TIME;
	END_VAR
	VAR_OUTPUT
		sDateTime : STRING[19];
	END_VAR
	VAR
		_dtStruc : DTStructure;
		_s2dig : STRING[2];
		_b2dig : REFERENCE TO ARRAY[0..1] OF USINT;
	END_VAR
END_FUNCTION_BLOCK

FUNCTION_BLOCK mnParam_datetoa (*Wandelt Datum Zeit in ISO String*)
	VAR_INPUT
		dtTimestamp : DATE_AND_TIME;
	END_VAR
	VAR_OUTPUT
		sDate : STRING[11];
	END_VAR
	VAR
		_dtStruc : DTStructure;
		_s2dig : STRING[2];
		_b2dig : REFERENCE TO ARRAY[0..1] OF USINT;
	END_VAR
END_FUNCTION_BLOCK

FUNCTION_BLOCK mnParam_WriteCSV253_Mem (*Versions Kopfzeile*)
	VAR_INPUT
		enable : BOOL;
		pMem : UDINT;
		lMaxSize : UDINT;
		VersionRow : mnParam_HeaderVersionRow_typ;
	END_VAR
	VAR_OUTPUT
		status : UINT;
	END_VAR
	VAR_IN_OUT
		lSize : UDINT;
	END_VAR
	VAR
		_pUtfString : REFERENCE TO ARRAY[0..11] OF UINT;
		_sVersion : STRING[5];
		_lLen : UDINT;
		_dttoa : mnParam_datetimetoa;
	END_VAR
END_FUNCTION_BLOCK

FUNCTION_BLOCK mnParam_WriteCSV252_Mem (*Versions Kopfzeile*)
	VAR_INPUT
		enable : BOOL;
		pMem : UDINT;
		lMaxSize : UDINT;
		MachineNoRow : mnParam_HeaderMachineNoRow_typ;
	END_VAR
	VAR_OUTPUT
		status : UINT;
	END_VAR
	VAR_IN_OUT
		lSize : UDINT;
	END_VAR
	VAR
		_pUtfString : REFERENCE TO ARRAY[0..11] OF UINT;
		_lLen : UDINT;
	END_VAR
END_FUNCTION_BLOCK

FUNCTION_BLOCK mnParam_WriteCSV251_Mem (*Dateizeitstempel schreiben*)
	VAR_INPUT
		enable : BOOL;
		pMem : UDINT;
		lMaxSize : UDINT;
		TimeRow : mnParam_HeaderTimeRow_typ;
	END_VAR
	VAR_OUTPUT
		status : UINT;
	END_VAR
	VAR_IN_OUT
		lSize : UDINT;
	END_VAR
	VAR
		_pUtfString : REFERENCE TO ARRAY[0..11] OF UINT;
		_dttoa : mnParam_datetimetoa;
	END_VAR
END_FUNCTION_BLOCK

FUNCTION_BLOCK mnParam_WriteCSV10_Mem (*Datenzeile numerisch schreiben*)
	VAR_INPUT
		enable : BOOL;
		pMem : UDINT;
		lMaxSize : UDINT;
		NumRow : mnParam_CsvNumRow_typ;
	END_VAR
	VAR_OUTPUT
		status : UINT;
	END_VAR
	VAR_IN_OUT
		lSize : UDINT;
	END_VAR
	VAR
		_pUtfString : REFERENCE TO ARRAY[0..11] OF UINT;
		_sNumeric : STRING[11];
		_lLen : UDINT;
	END_VAR
END_FUNCTION_BLOCK

FUNCTION_BLOCK mnParam_WriteCSV20_Mem (*String Daten schreiben*)
	VAR_INPUT
		enable : BOOL;
		pMem : UDINT;
		lMaxSize : UDINT;
		StringRow : mnParam_CsvStringRow_typ;
	END_VAR
	VAR_OUTPUT
		status : UINT;
	END_VAR
	VAR_IN_OUT
		lSize : UDINT;
	END_VAR
	VAR
		_pUtfString : REFERENCE TO ARRAY[0..11] OF UINT;
		_sNumeric : STRING[11];
		_lLen : UDINT;
	END_VAR
END_FUNCTION_BLOCK

FUNCTION_BLOCK mnParam_WriteCSV80_Mem (*String Daten schreiben*)
	VAR_INPUT
		enable : BOOL;
		pMem : UDINT;
		lMaxSize : UDINT;
		ContentRow : mnParam_CsvContent_typ;
	END_VAR
	VAR_OUTPUT
		status : UINT;
	END_VAR
	VAR_IN_OUT
		lSize : UDINT;
	END_VAR
	VAR
		_pUtfString : REFERENCE TO ARRAY[0..15] OF UINT;
		_sValue : STRING[11];
		_lLen : UDINT;
		_dttoa : mnParam_datetimetoa;
	END_VAR
END_FUNCTION_BLOCK

FUNCTION_BLOCK mnParam_WriteCSV81_Mem (*String Daten schreiben*)
	VAR_INPUT
		enable : BOOL;
		pMem : UDINT;
		lMaxSize : UDINT;
		CPRow : mnParam_CProw_typ;
	END_VAR
	VAR_OUTPUT
		status : UINT;
	END_VAR
	VAR_IN_OUT
		lSize : UDINT;
	END_VAR
	VAR
		_pUtfString : REFERENCE TO ARRAY[0..15] OF UINT;
		_sValue : STRING[23];
		_lLen : UDINT;
		_dttoa : mnParam_datetimetoa;
	END_VAR
END_FUNCTION_BLOCK

FUNCTION_BLOCK mnParam_WriteCSV90_Mem (*String Daten schreiben*)
	VAR_INPUT
		enable : BOOL;
		pMem : UDINT;
		lMaxSize : UDINT;
		IPRow : mnParam_CsvIPRow_typ;
	END_VAR
	VAR_OUTPUT
		status : UINT;
	END_VAR
	VAR_IN_OUT
		lSize : UDINT;
	END_VAR
	VAR
		_pUtfString : REFERENCE TO ARRAY[0..15] OF UINT;
		_lLen : UDINT;
	END_VAR
END_FUNCTION_BLOCK

FUNCTION_BLOCK mnParam_WriteCSV11_Mem (*Datenzeile numerisch schreiben*)
	VAR_INPUT
		enable : BOOL;
		pMem : UDINT;
		lMaxSize : UDINT;
		NumRow : mnParam_CsvNumRow_typ;
	END_VAR
	VAR_OUTPUT
		status : UINT;
	END_VAR
	VAR_IN_OUT
		lSize : UDINT;
	END_VAR
	VAR
		_pUtfString : REFERENCE TO ARRAY[0..11] OF UINT;
		_sNumeric : STRING[31];
		_lLen : UDINT;
		_pdiValue : REFERENCE TO DINT;
		_rValue : REAL;
	END_VAR
END_FUNCTION_BLOCK
```

#### mnParamLib-History.txt
```
0.01.0	AH: Erste Version für Landshut

0.02.0  AH: Erweiterung um REAL-Parameter

0.07.0	AH: CSV-Zeilen 80, 200, 210 und 248 ergänzt
```

#### mnParam_BinarySearchInNumeric.st
```iecst
(********************************************************************
 * COPYRIGHT -- Microsoft
 ********************************************************************
 * Library: BinSearch
 * File: BinarySearchInNumeric.st
 * Author: Reese_Markus
 * Created: July 25, 2011
 ********************************************************************
 * Implementation of library BinSearch
 ********************************************************************)

(* TODO: Add your comment here *)
FUNCTION_BLOCK mnParam_BinarySearchInNumeric

IF enable THEN

	IF lpList = 0 OR lMaxRow < 1 THEN
		// Null-Pointer
		status := 1;
		RETURN;
	END_IF

	// Access auf dynamische Struktur
	_CsvStructNumDyn ACCESS lpList;

	_lMin := 1;
	_lMax := lMaxRow;

	WHILE TRUE DO

		IF (_lMin <= _lMax) THEN

			// Suche nach korrektem IdxPar
			// Middle Index berechnen
			_lMid := (_lMin + _lMax) / 2;

			// Suche erfolgreich?
			IF (CsvStructNum.wIdxNumPar = _CsvStructNumDyn.CsvNum[_lMid].wIdxNumPar) THEN
				// korrekten IdxPar gefunden

				// Suche erfolgreich?
				IF (CsvStructNum.wArrIdx1 = _CsvStructNumDyn.CsvNum[_lMid].wArrIdx1) THEN
					// korrekten wArrIdx1 gefunden

					// Suche erfolgreich?
					IF (CsvStructNum.wArrIdx2 = _CsvStructNumDyn.CsvNum[_lMid].wArrIdx2) THEN
						// korrekten wArrIdx2 gefunden

						// Suche erfolgreich?
						IF (CsvStructNum.wArrIdx3 = _CsvStructNumDyn.CsvNum[_lMid].wArrIdx3) THEN
							// korrekten wArrIdx3 gefunden

							// Suche erfolgreich?
							IF (CsvStructNum.wArrIdx4 = _CsvStructNumDyn.CsvNum[_lMid].wArrIdx4) THEN
								// korrekten wArrIdx4 gefunden

								// gefundenen Zeilen Index übergeben
								lFoundRow := _lMid;

								status := 0; // ohne Fehler durchlaufen

								EXIT; // While-Schleife der Suche verlassen

							ELSIF (CsvStructNum.wArrIdx4 < _CsvStructNumDyn.CsvNum[_lMid].wArrIdx4) THEN
								// gefundener Index ist grösser
								_lMax := _lMid - 1;
							ELSE
								// gefundener Index ist kleiner
								_lMin := _lMid + 1;
							END_IF;

						ELSIF (CsvStructNum.wArrIdx3 < _CsvStructNumDyn.CsvNum[_lMid].wArrIdx3) THEN
							// gefundener Index ist grösser
							_lMax := _lMid - 1;
						ELSE
							// gefundener Index ist kleiner
							_lMin := _lMid + 1;
						END_IF;

					ELSIF (CsvStructNum.wArrIdx2 < _CsvStructNumDyn.CsvNum[_lMid].wArrIdx2) THEN
						// gefundener Index ist grösser
						_lMax := _lMid - 1;
					ELSE
						// gefundener Index ist kleiner
						_lMin := _lMid + 1;
					END_IF;

				ELSIF (CsvStructNum.wArrIdx1 < _CsvStructNumDyn.CsvNum[_lMid].wArrIdx1) THEN
					// gefundener Index ist grösser
					_lMax := _lMid - 1;
				ELSE
					// gefundener Index ist kleiner
					_lMin := _lMid + 1;
				END_IF;

			ELSIF (CsvStructNum.wIdxNumPar < _CsvStructNumDyn.CsvNum[_lMid].wIdxNumPar) THEN
				// gefundener Index ist grösser
				_lMax := _lMid - 1;
			ELSE
				// gefundener Index ist kleiner
				_lMin := _lMid + 1;
			END_IF;

		ELSIF (_lMin > _lMax) THEN
			// Fehler in der Binären-Suche
			// zB entsprechende Zeile konnte nicht gefunden werden
			status := 2;
			EXIT;
		END_IF;

	END_WHILE;

ELSE

	status := 65534; // Eingang enable nicht gesetzt

END_IF

END_FUNCTION_BLOCK
```

#### mnParam_BinarySearchInString.st - Binärsuche von CSV-String-Container-Zeilen
```iecst
(********************************************************************
 * COPYRIGHT -- Microsoft
 ********************************************************************
 * Library: mnParamLib
 * File: mnParam_BinarySearchInString.st
 * Author: hunholz
 * Created: August 01, 2011
 ********************************************************************
 * Implementation of library mnParamLib
 ********************************************************************)

(* Binärsuche von CSV-String-Container-Zeilen *)
FUNCTION_BLOCK mnParam_BinarySearchInString

IF enable THEN

	IF lpList = 0 OR lMaxRow < 1 THEN
		// Null-Pointer
		status := 1;
		RETURN;
	END_IF

	// Access auf dynamische Struktur
	_CsvStructStringDyn ACCESS lpList;

	_lMin := 1;
	_lMax := lMaxRow;

	WHILE TRUE DO

		IF (_lMin <= _lMax) THEN

			// Suche nach korrektem IdxPar
			// Middle Index berechnen
			_lMid := (_lMin + _lMax) / 2;

			// Suche erfolgreich?
			IF (CsvStructString.wIdxStringPar = _CsvStructStringDyn.CsvString[_lMid].wIdxStringPar) THEN
				// korrekten IdxPar gefunden

				// Suche erfolgreich?
				IF (CsvStructString.wArrIdx1 = _CsvStructStringDyn.CsvString[_lMid].wArrIdx1) THEN
					// korrekten wArrIdx1 gefunden

					// Suche erfolgreich?
					IF (CsvStructString.wArrIdx2 = _CsvStructStringDyn.CsvString[_lMid].wArrIdx2) THEN
						// korrekten wArrIdx2 gefunden

						// Suche erfolgreich?
						IF (CsvStructString.wArrIdx3 = _CsvStructStringDyn.CsvString[_lMid].wArrIdx3) THEN
							// korrekten wArrIdx3 gefunden

							// Suche erfolgreich?
							IF (CsvStructString.wArrIdx4 = _CsvStructStringDyn.CsvString[_lMid].wArrIdx4) THEN
								// korrekten wArrIdx4 gefunden

								// gefundenen Zeilen Index übergeben
								lFoundRow := _lMid;

								status := 0; // ohne Fehler durchlaufen

								EXIT; // While-Schleife der Suche verlassen

							ELSIF (CsvStructString.wArrIdx4 < _CsvStructStringDyn.CsvString[_lMid].wArrIdx4) THEN
								// gefundener Index ist grösser
								_lMax := _lMid - 1;
							ELSE
								// gefundener Index ist kleiner
								_lMin := _lMid + 1;
							END_IF;

						ELSIF (CsvStructString.wArrIdx3 < _CsvStructStringDyn.CsvString[_lMid].wArrIdx3) THEN
							// gefundener Index ist grösser
							_lMax := _lMid - 1;
						ELSE
							// gefundener Index ist kleiner
							_lMin := _lMid + 1;
						END_IF;

					ELSIF (CsvStructString.wArrIdx2 < _CsvStructStringDyn.CsvString[_lMid].wArrIdx2) THEN
						// gefundener Index ist grösser
						_lMax := _lMid - 1;
					ELSE
						// gefundener Index ist kleiner
						_lMin := _lMid + 1;
					END_IF;

				ELSIF (CsvStructString.wArrIdx1 < _CsvStructStringDyn.CsvString[_lMid].wArrIdx1) THEN
					// gefundener Index ist grösser
					_lMax := _lMid - 1;
				ELSE
					// gefundener Index ist kleiner
					_lMin := _lMid + 1;
				END_IF;

			ELSIF (CsvStructString.wIdxStringPar < _CsvStructStringDyn.CsvString[_lMid].wIdxStringPar) THEN
				// gefundener Index ist grösser
				_lMax := _lMid - 1;
			ELSE
				// gefundener Index ist kleiner
				_lMin := _lMid + 1;
			END_IF;

		ELSIF (_lMin > _lMax) THEN
			// Fehler in der Binären-Suche
			// zB entsprechende Zeile konnte nicht gefunden werden
			status := 2;
			EXIT;
		END_IF;

	END_WHILE;

ELSE

	status := 65534; // Eingang enable nicht gesetzt

END_IF

END_FUNCTION_BLOCK
```

#### mnParam_CountLines.st - Zählt die gültigen Zeilen der Datei und gibt eine Zeilenstruktur zurück
```iecst
(********************************************************************
 * COPYRIGHT -- Microsoft
 ********************************************************************
 * Library: mnParamLib
 * File: mnParam_CountLines.st
 * Author: hunholz
 * Created: July 25, 2011
 ********************************************************************
 * Implementation of library mnParamLib
 ********************************************************************)

(* Zählt die gültigen Zeilen der Datei und gibt eine Zeilenstruktur zurück *)
FUNCTION_BLOCK mnParam_CountLines

	IF enable THEN

		// Gültigkeit der Übergabeparameter
		IF pAdresses = 0 OR pLens = 0 OR MaxLines > 20000 OR pFile = 0 THEN
			status := 1;
			RETURN;
		END_IF

		status := 0;

		CntLines := 0;

		brsmemset(pAdresses, 0, UINT_TO_UDINT(MaxLines) * 4);
		brsmemset(pLens, 0, UINT_TO_UDINT(MaxLines) * 2);

		_plAdresses ACCESS pAdresses;
		_pwLens ACCESS pLens;

		_xNewLine := TRUE;

		FOR _p := pFile TO pFile + FileSize  - 2 BY 2 DO

			_pChar	ACCESS _p;

			IF _pChar = 16#000D OR _pChar = 16#000A THEN

				IF NOT _xNewLine THEN

					// Zeilenende gefunden
					_lDif := _p - _plAdresses[CntLines];

					_pwLens[CntLines] := UDINT_TO_UINT( (_lDif) / 2 );

				END_IF

				_xNewLine := TRUE;

				IF CntLines >= MaxLines THEN
					EXIT;
				END_IF

			ELSIF _xNewLine THEN

				CntLines := CntLines + 1;
				_plAdresses[CntLines]	:= _p;
				_xNewLine := FALSE;

			END_IF

		END_FOR

		IF NOT _xNewLine THEN

			_lDif := _p - _plAdresses[CntLines];

			_pwLens[CntLines] := UDINT_TO_UINT( (_lDif) / 2 );

		END_IF

	ELSE

		status := ERR_FUB_ENABLE_FALSE;

	END_IF

END_FUNCTION_BLOCK
```
